KUKA KRL program: MyProgram_162().src

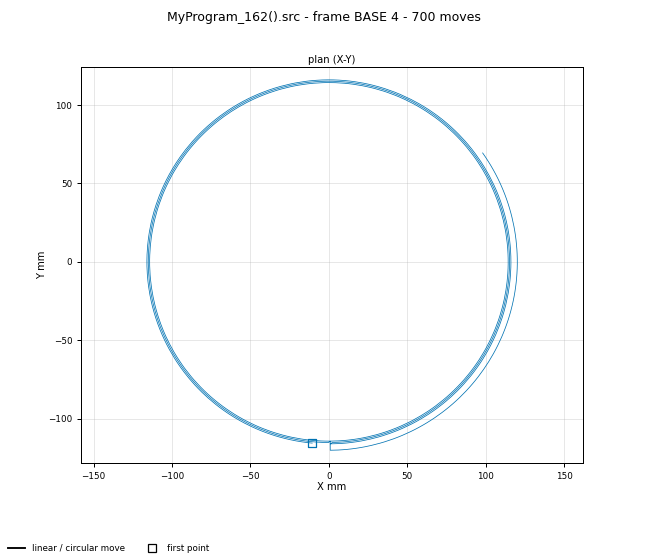
[picture p0: tool path of MyProgram_162().src in frame BASE 4, 700 of 700 moves have a stored position in this frame; points joined in program order, loops and branches not executed]
&ACCESS RVP
&REL 1
&PARAM TEMPLATE = C:\KRC\Roboter\Template\vorgabe
&PARAM EDITMASK = *
DEF MyProgram_162()
; ---- Setting reference (Base) ----
$BASE = BASE_DATA[4]

; --------------------------
; ---- Setting tool (TCP) ----
$TOOL = TOOL_DATA[3]
; --------------------------

$VEL.CP = VEL_APROX_PRINT
Startdeposition()
$VEL.CP = VEL_PRINT
LIN {X -10.6653,Y -115.559,Z 123,A -99.1684,B 24.9575,C -1.5067,E1 24.9847,E2 185.24} C_DIS
LIN {X -13.6922,Y -115.2397,Z 123,A -100.788,B 24.9577,C -1.5018,E1 24.9802,E2 186.8723} C_DIS
LIN {X -17.6034,Y -114.7073,Z 123,A -102.6994,B 24.9577,C -1.5039,E1 24.9749,E2 188.7803} C_DIS
LIN {X -20.9745,Y -114.1398,Z 123,A -104.185,B 24.9571,C -1.5133,E1 24.9709,E2 190.2451} C_DIS
LIN {X -25.0062,Y -113.3242,Z 123,A -106.7407,B 24.9583,C -1.4914,E1 24.9637,E2 192.8559} C_DIS
LIN {X -28.1463,Y -112.5871,Z 123,A -108.1226,B 24.9578,C -1.5013,E1 24.96,E2 194.216} C_DIS
LIN {X -31.7748,Y -111.6155,Z 123,A -109.9543,B 24.9576,C -1.5036,E1 24.9551,E2 196.0454} C_DIS
LIN {X -34.7534,Y -110.7249,Z 123,A -111.6242,B 24.9579,C -1.4989,E1 24.9506,E2 197.7293} C_DIS
LIN {X -38.9895,Y -109.306,Z 123,A -113.7372,B 24.9576,C -1.5047,E1 24.9451,E2 199.8326} C_DIS
LIN {X -42.4675,Y -108.0007,Z 123,A -115.4677,B 24.9572,C -1.5109,E1 24.9406,E2 201.5519} C_DIS
LIN {X -45.3067,Y -106.841,Z 123,A -117.0721,B 24.9574,C -1.5086,E1 24.9364,E2 203.1654} C_DIS
LIN {X -48.6937,Y -105.3407,Z 123,A -118.8003,B 24.957,C -1.515,E1 24.9321,E2 204.8826} C_DIS
LIN {X -53.8437,Y -102.8035,Z 123,A -121.6909,B 24.957,C -1.5162,E1 24.9249,E2 207.7782} C_DIS
LIN {X -57.1329,Y -101.0142,Z 123,A -124.0798,B 24.9581,C -1.4959,E1 24.9189,E2 210.2222} C_DIS
LIN {X -60.7707,Y -98.8681,Z 123,A -125.684,B 24.9568,C -1.5193,E1 24.9152,E2 211.7758} C_DIS
LIN {X -63.696,Y -97.0077,Z 123,A -127.252,B 24.9563,C -1.5281,E1 24.9115,E2 213.328} C_DIS
LIN {X -66.3521,Y -95.2106,Z 123,A -128.9266,B 24.9563,C -1.5268,E1 24.9077,E2 215.0111} C_DIS
LIN {X -69.3236,Y -93.0704,Z 123,A -130.8195,B 24.9563,C -1.5264,E1 24.9034,E2 216.9117} C_DIS
LIN {X -71.8676,Y -91.1191,Z 123,A -133.4324,B 24.9586,C -1.4866,E1 24.8975,E2 219.629} C_DIS
LIN {X -77.0205,Y -86.8086,Z 123,A -135.5024,B 24.9553,C -1.5447,E1 24.8934,E2 221.5689} C_DIS
LIN {X -81.0208,Y -83.0887,Z 123,A -138.4564,B 24.9556,C -1.5395,E1 24.8873,E2 224.5473} C_DIS
LIN {X -83.5609,Y -80.5308,Z 123,A -140.1615,B 24.9552,C -1.5465,E1 24.884,E2 226.2431} C_DIS
LIN {X -85.4663,Y -78.5057,Z 123,A -142.2929,B 24.9568,C -1.5184,E1 24.8799,E2 228.4508} C_DIS
LIN {X -88.8943,Y -74.604,Z 123,A -143.9688,B 24.9544,C -1.5609,E1 24.877,E2 230.0333} C_DIS
LIN {X -92.3379,Y -70.2979,Z 123,A -146.9806,B 24.9547,C -1.5555,E1 24.8717,E2 233.0722} C_DIS
LIN {X -94.5964,Y -67.2251,Z 123,A -148.7888,B 24.9542,C -1.5633,E1 24.8688,E2 234.8705} C_DIS
LIN {X -96.8103,Y -63.9955,Z 123,A -150.6696,B 24.9538,C -1.5704,E1 24.8658,E2 236.7437} C_DIS
LIN {X -98.2369,Y -61.784,Z 123,A -152.1414,B 24.954,C -1.5668,E1 24.8636,E2 238.2317} C_DIS
LIN {X -100.5513,Y -57.9404,Z 123,A -153.9732,B 24.9527,C -1.5884,E1 24.8611,E2 240.0214} C_DIS
LIN {X -101.7139,Y -55.8775,Z 123,A -155.4383,B 24.9533,C -1.5795,E1 24.859,E2 241.5155} C_DIS
LIN {X -103.2771,Y -52.9291,Z 123,A -157.0466,B 24.9529,C -1.5857,E1 24.857,E2 243.1175} C_DIS
LIN {X -104.6961,Y -50.0641,Z 123,A -158.8223,B 24.9531,C -1.5822,E1 24.8548,E2 244.9113} C_DIS
LIN {X -106.1854,Y -46.8231,Z 123,A -160.8908,B 24.9535,C -1.5748,E1 24.8524,E2 247.0087} C_DIS
LIN {X -107.7171,Y -43.1859,Z 123,A -162.4847,B 24.9523,C -1.5948,E1 24.8508,E2 248.5638} C_DIS
LIN {X -109.095,Y -39.5722,Z 123,A -164.3294,B 24.9518,C -1.6031,E1 24.849,E2 250.3991} C_DIS
LIN {X -110.3696,Y -35.8636,Z 123,A -166.2617,B 24.9515,C -1.6091,E1 24.8473,E2 252.328} C_DIS
LIN {X -111.5262,Y -32.0901,Z 123,A -168.0218,B 24.9507,C -1.6227,E1 24.8459,E2 254.0659} C_DIS
LIN {X -112.5763,Y -28.1905,Z 123,A -170.1776,B 24.9507,C -1.6223,E1 24.8444,E2 256.2354} C_DIS
LIN {X -113.2511,Y -25.3421,Z 123,A -171.5538,B 24.9502,C -1.6296,E1 24.8435,E2 257.6022} C_DIS
LIN {X -114.1339,Y -21.0071,Z 123,A -174.7127,B 24.9522,C -1.5975,E1 24.8418,E2 260.8563} C_DIS
LIN {X -115.0069,Y -15.5386,Z 123,A -176.6028,B 24.9496,C -1.6399,E1 24.8411,E2 262.6566} C_DIS
LIN {X -115.4108,Y -12.1655,Z 123,A -178.893,B 24.9508,C -1.6208,E1 24.8404,E2 265.006} C_DIS
LIN {X -115.7852,Y -7.8379,Z 123,A 178.8146,B 24.9508,C -1.6219,E1 24.84,E2 267.3096} C_DIS
LIN {X -116.0178,Y -2.8199,Z 123,A 176.9216,B 24.9488,C -1.6533,E1 24.8398,E2 269.1392} C_DIS
LIN {X -116.0475,Y 0.856,Z 123,A 174.7066,B 24.9494,C -1.6433,E1 24.8398,E2 271.3915} C_DIS
LIN {X -115.9508,Y 4.8049,Z 123,A 172.4484,B 24.9498,C -1.6374,E1 24.8401,E2 273.6772} C_DIS
LIN {X -115.6096,Y 10.1176,Z 123,A 170.5898,B 24.9473,C -1.6766,E1 24.8405,E2 275.4536} C_DIS
LIN {X -115.0956,Y 14.8542,Z 123,A 168.1879,B 24.947,C -1.6823,E1 24.8413,E2 277.8562} C_DIS
LIN {X -114.5033,Y 18.8864,Z 123,A 166.2109,B 24.9465,C -1.6902,E1 24.8421,E2 279.8261} C_DIS
LIN {X -113.9089,Y 22.1913,Z 123,A 164.4813,B 24.9463,C -1.6927,E1 24.843,E2 281.56} C_DIS
LIN {X -113.3762,Y 24.7683,Z 123,A 162.8897,B 24.9468,C -1.6852,E1 24.844,E2 283.1788} C_DIS
LIN {X -112.6272,Y 27.9821,Z 123,A 161.5978,B 24.9456,C -1.7039,E1 24.8448,E2 284.4338} C_DIS
LIN {X -111.4941,Y 32.2032,Z 123,A 159.3971,B 24.9453,C -1.7091,E1 24.8464,E2 286.6349} C_DIS
LIN {X -110.195,Y 36.4032,Z 123,A 156.9707,B 24.9455,C -1.7057,E1 24.8485,E2 289.0832} C_DIS
LIN {X -108.2506,Y 41.8313,Z 123,A 154.2761,B 24.9445,C -1.7207,E1 24.8511,E2 291.7574} C_DIS
LIN {X -106.9132,Y 45.1354,Z 123,A 152.6645,B 24.9438,C -1.7321,E1 24.8528,E2 293.3507} C_DIS
LIN {X -105.5414,Y 48.2602,Z 123,A 150.7928,B 24.9439,C -1.7297,E1 24.855,E2 295.2384} C_DIS
LIN {X -103.8814,Y 51.7333,Z 123,A 148.9469,B 24.9434,C -1.7376,E1 24.8572,E2 297.0754} C_DIS
LIN {X -101.8776,Y 55.5757,Z 123,A 146.1169,B 24.9448,C -1.7164,E1 24.8611,E2 299.971} C_DIS
LIN {X -99.431,Y 59.8444,Z 123,A 144.3767,B 24.9425,C -1.751,E1 24.8634,E2 301.6377} C_DIS
LIN {X -97.3709,Y 63.1413,Z 123,A 141.7758,B 24.944,C -1.7291,E1 24.8675,E2 304.3039} C_DIS
LIN {X -94.7272,Y 67.0417,Z 123,A 140.3014,B 24.9413,C -1.7698,E1 24.8697,E2 305.6885} C_DIS
LIN {X -91.4771,Y 71.4147,Z 123,A 137.3922,B 24.9414,C -1.7682,E1 24.8746,E2 308.6155} C_DIS
LIN {X -87.1641,Y 76.6172,Z 123,A 133.5732,B 24.9421,C -1.7574,E1 24.8816,E2 312.4776} C_DIS
LIN {X -84.599,Y 79.4396,Z 123,A 132.0333,B 24.9409,C -1.7761,E1 24.8844,E2 313.9799} C_DIS
LIN {X -82.0963,Y 82.026,Z 123,A 130.4546,B 24.94,C -1.7885,E1 24.8875,E2 315.5358} C_DIS
LIN {X -79.8971,Y 84.1676,Z 123,A 128.9268,B 24.9398,C -1.7916,E1 24.8905,E2 317.0624} C_DIS
LIN {X -77.5135,Y 86.3673,Z 123,A 127.1384,B 24.9401,C -1.7877,E1 24.8943,E2 318.8673} C_DIS
LIN {X -73.9241,Y 89.4593,Z 123,A 124.9854,B 24.9392,C -1.8006,E1 24.8988,E2 320.9979} C_DIS
LIN {X -72.0186,Y 90.9998,Z 123,A 123.6847,B 24.9393,C -1.7996,E1 24.9017,E2 322.306} C_DIS
LIN {X -69.5493,Y 92.9008,Z 123,A 122.1969,B 24.9389,C -1.8049,E1 24.9049,E2 323.7865} C_DIS
LIN {X -66.4177,Y 95.165,Z 123,A 120.2261,B 24.9389,C -1.8062,E1 24.9094,E2 325.761} C_DIS
LIN {X -64.3163,Y 96.5987,Z 123,A 118.456,B 24.9401,C -1.7876,E1 24.9137,E2 327.5813} C_DIS
LIN {X -61.0227,Y 98.7123,Z 123,A 116.9584,B 24.9387,C -1.8091,E1 24.9171,E2 329.0325} C_DIS
LIN {X -57.9117,Y 100.5678,Z 123,A 115.2449,B 24.9382,C -1.8154,E1 24.9212,E2 330.736} C_DIS
LIN {X -54.6063,Y 102.4019,Z 123,A 113.3425,B 24.9382,C -1.8171,E1 24.9259,E2 332.6397} C_DIS
LIN {X -51.6065,Y 103.9443,Z 123,A 111.7134,B 24.9378,C -1.8214,E1 24.9299,E2 334.263} C_DIS
LIN {X -49.021,Y 105.1883,Z 123,A 110.011,B 24.9385,C -1.8117,E1 24.9343,E2 335.9928} C_DIS
LIN {X -45.1475,Y 106.9081,Z 123,A 108.1625,B 24.9376,C -1.825,E1 24.939,E2 337.8141} C_DIS
LIN {X -42.56,Y 107.9644,Z 123,A 106.5783,B 24.938,C -1.8183,E1 24.9431,E2 339.4176} C_DIS
LIN {X -38.4699,Y 109.4884,Z 123,A 104.5881,B 24.9374,C -1.828,E1 24.9483,E2 341.3887} C_DIS
LIN {X -34.7829,Y 110.7157,Z 123,A 102.1474,B 24.9387,C -1.8084,E1 24.9549,E2 343.8804} C_DIS
LIN {X -30.8214,Y 111.8839,Z 123,A 100.7644,B 24.9367,C -1.8382,E1 24.9585,E2 345.1949} C_DIS
LIN {X -24.2525,Y 113.4886,Z 123,A 97.3058,B 24.9368,C -1.8362,E1 24.9679,E2 348.6629} C_DIS
LIN {X -21.2452,Y 114.0905,Z 123,A 94.6996,B 24.9399,C -1.7914,E1 24.9754,E2 351.3782} C_DIS
LIN {X -14.8714,Y 115.0933,Z 123,A 92.6352,B 24.9365,C -1.8408,E1 24.9807,E2 353.3269} C_DIS
LIN {X -11.5372,Y 115.4765,Z 123,A 90.862,B 24.9368,C -1.8367,E1 24.9857,E2 355.111} C_DIS
LIN {X -7.9886,Y 115.775,Z 123,A 89.1698,B 24.9365,C -1.8403,E1 24.9904,E2 356.7953} C_DIS
LIN {X -4.2713,Y 115.9737,Z 123,A 87.2428,B 24.9367,C -1.8371,E1 24.9958,E2 358.7304} C_DIS
LIN {X -0.6516,Y 116.0483,Z 123,A 85.579,B 24.9363,C -1.8429,E1 25.0004,E2 360.3805} C_DIS
LIN {X 2.8366,Y 116.0176,Z 123,A 83.7142,B 24.9368,C -1.8369,E1 25.0056,E2 362.2592} C_DIS
LIN {X 6.415,Y 115.8727,Z 123,A 82.0622,B 24.9364,C -1.8421,E1 25.0102,E2 363.8985} C_DIS
LIN {X 10.0554,Y 115.6153,Z 123,A 80.1581,B 24.9367,C -1.8375,E1 25.0155,E2 365.8124} C_DIS
LIN {X 13.4144,Y 115.2723,Z 123,A 78.5907,B 24.9364,C -1.8416,E1 25.0198,E2 367.3691} C_DIS
LIN {X 16.9015,Y 114.8143,Z 123,A 76.9179,B 24.9363,C -1.8439,E1 25.0244,E2 369.0349} C_DIS
LIN {X 22.1519,Y 113.9165,Z 123,A 73.8926,B 24.9375,C -1.8256,E1 25.0329,E2 372.1002} C_DIS
LIN {X 25.3525,Y 113.2488,Z 123,A 72.6719,B 24.9364,C -1.842,E1 25.0361,E2 373.2804} C_DIS
LIN {X 28.1703,Y 112.5796,Z 123,A 71.0663,B 24.937,C -1.8335,E1 25.0405,E2 374.904} C_DIS
LIN {X 31.8716,Y 111.5881,Z 123,A 69.1035,B 24.9373,C -1.829,E1 25.0458,E2 376.874} C_DIS
LIN {X 35.8448,Y 110.3757,Z 123,A 67.2411,B 24.9368,C -1.8358,E1 25.0507,E2 378.717} C_DIS
LIN {X 39.5647,Y 109.0977,Z 123,A 65.5874,B 24.9361,C -1.8468,E1 25.055,E2 380.3412} C_DIS
LIN {X 41.7509,Y 108.2819,Z 123,A 64.0219,B 24.9374,C -1.8273,E1 25.0592,E2 381.9496} C_DIS
LIN {X 45.319,Y 106.8358,Z 123,A 62.2201,B 24.9372,C -1.8297,E1 25.0638,E2 383.7415} C_DIS
LIN {X 52.4206,Y 103.537,Z 123,A 58.4693,B 24.9372,C -1.8301,E1 25.0733,E2 387.4816} C_DIS
LIN {X 57.4012,Y 100.8611,Z 123,A 55.567,B 24.9378,C -1.8212,E1 25.0804,E2 390.3965} C_DIS
LIN {X 60.4595,Y 99.0572,Z 123,A 53.8305,B 24.938,C -1.8194,E1 25.0845,E2 392.1321} C_DIS
LIN {X 63.7326,Y 96.9836,Z 123,A 51.8571,B 24.9384,C -1.8136,E1 25.0892,E2 394.1127} C_DIS
LIN {X 67.2845,Y 94.5539,Z 123,A 49.7895,B 24.9384,C -1.8125,E1 25.0939,E2 396.1757} C_DIS
LIN {X 69.3854,Y 93.024,Z 123,A 48.1836,B 24.9396,C -1.7956,E1 25.0976,E2 397.8157} C_DIS
LIN {X 72.0684,Y 90.9604,Z 123,A 46.557,B 24.9396,C -1.7945,E1 25.1011,E2 399.4389} C_DIS
LIN {X 74.6917,Y 88.8214,Z 123,A 45.1593,B 24.939,C -1.8037,E1 25.1041,E2 400.8096} C_DIS
LIN {X 77.4628,Y 86.4127,Z 123,A 43.4207,B 24.939,C -1.8035,E1 25.1077,E2 402.5419} C_DIS
LIN {X 80.3599,Y 83.7256,Z 123,A 41.486,B 24.9393,C -1.8001,E1 25.1116,E2 404.4764} C_DIS
LIN {X 82.6619,Y 81.4535,Z 123,A 39.6068,B 24.9404,C -1.7837,E1 25.1154,E2 406.3864} C_DIS
LIN {X 86.7428,Y 77.094,Z 123,A 36.8843,B 24.9401,C -1.7874,E1 25.1205,E2 409.0882} C_DIS
LIN {X 88.767,Y 74.7562,Z 123,A 35.3125,B 24.9405,C -1.7817,E1 25.1234,E2 410.6664} C_DIS
LIN {X 91.1283,Y 71.856,Z 123,A 33.585,B 24.9405,C -1.7828,E1 25.1263,E2 412.3833} C_DIS
LIN {X 93.4714,Y 68.7808,Z 123,A 31.6666,B 24.9408,C -1.7776,E1 25.1296,E2 414.3048} C_DIS
LIN {X 96.8913,Y 63.8727,Z 123,A 28.7323,B 24.9412,C -1.7709,E1 25.1342,E2 417.2404} C_DIS
LIN {X 99.1052,Y 60.3806,Z 123,A 26.9313,B 24.9408,C -1.7766,E1 25.1368,E2 419.0188} C_DIS
LIN {X 102.1738,Y 55.0296,Z 123,A 23.7699,B 24.9418,C -1.7628,E1 25.1412,E2 422.1963} C_DIS
LIN {X 105.2146,Y 48.9644,Z 123,A 20.4053,B 24.9424,C -1.7526,E1 25.1454,E2 425.567} C_DIS
LIN {X 106.7262,Y 45.5792,Z 123,A 18.5385,B 24.9429,C -1.7456,E1 25.1475,E2 427.4402} C_DIS
LIN {X 108.0181,Y 42.4232,Z 123,A 16.8907,B 24.9431,C -1.7423,E1 25.1492,E2 429.0866} C_DIS
LIN {X 109.3788,Y 38.7822,Z 123,A 14.9282,B 24.9436,C -1.7345,E1 25.1511,E2 431.0564} C_DIS
LIN {X 110.9984,Y 33.8711,Z 123,A 12.5513,B 24.9436,C -1.735,E1 25.1531,E2 433.4187} C_DIS
LIN {X 112.1204,Y 29.9461,Z 123,A 10.2332,B 24.9449,C -1.7146,E1 25.1549,E2 435.7716} C_DIS
LIN {X 113.1662,Y 25.7141,Z 123,A 8.2717,B 24.9448,C -1.7168,E1 25.1561,E2 437.7166} C_DIS
LIN {X 114.1323,Y 21.0161,Z 123,A 5.995,B 24.945,C -1.7136,E1 25.1573,E2 439.9875} C_DIS
LIN {X 114.678,Y 17.793,Z 123,A 4.3378,B 24.9454,C -1.7065,E1 25.1581,E2 441.6518} C_DIS
LIN {X 115.2213,Y 13.8498,Z 123,A 2.4673,B 24.9455,C -1.7046,E1 25.1588,E2 443.5156} C_DIS
LIN {X 115.5668,Y 10.5813,Z 123,A 0.8306,B 24.9459,C -1.6987,E1 25.1592,E2 445.1565} C_DIS
LIN {X 115.8416,Y 6.9777,Z 123,A -1.0576,B 24.9466,C -1.688,E1 25.1596,E2 447.0588} C_DIS
LIN {X 115.9975,Y 3.4945,Z 123,A -2.7088,B 24.9467,C -1.6858,E1 25.1597,E2 448.7055} C_DIS
LIN {X 116.0499,Y -0.4908,Z 123,A -4.6581,B 24.9471,C -1.6802,E1 25.1597,E2 450.6564} C_DIS
LIN {X 115.993,Y -3.6417,Z 123,A -6.2118,B 24.9474,C -1.6752,E1 25.1597,E2 452.2125} C_DIS
LIN {X 115.8011,Y -7.6013,Z 123,A -8.1306,B 24.9477,C -1.6706,E1 25.1594,E2 454.1307} C_DIS
LIN {X 115.5426,Y -10.843,Z 123,A -9.6833,B 24.9479,C -1.6679,E1 25.159,E2 455.6807} C_DIS
LIN {X 115.1957,Y -14.0682,Z 123,A -11.4618,B 24.9487,C -1.6543,E1 25.1584,E2 457.4807} C_DIS
LIN {X 114.3495,Y -19.8061,Z 123,A -14.2853,B 24.9492,C -1.6468,E1 25.1572,E2 460.3052} C_DIS
LIN {X 112.7554,Y -27.4564,Z 123,A -17.8097,B 24.949,C -1.6502,E1 25.1552,E2 463.8013} C_DIS
LIN {X 111.5256,Y -32.092,Z 123,A -20.3392,B 24.9499,C -1.6349,E1 25.1533,E2 466.3523} C_DIS
LIN {X 110.4511,Y -35.6117,Z 123,A -22.9008,B 24.9524,C -1.5941,E1 25.151,E2 468.9954} C_DIS
LIN {X 108.7581,Y -40.4935,Z 123,A -24.807,B 24.951,C -1.6163,E1 25.1493,E2 470.8387} C_DIS
LIN {X 107.4122,Y -43.9351,Z 123,A -26.5091,B 24.951,C -1.6164,E1 25.1475,E2 472.5311} C_DIS
LIN {X 106.4459,Y -46.2269,Z 123,A -28.2646,B 24.9528,C -1.5878,E1 25.1455,E2 474.3443} C_DIS
LIN {X 104.71,Y -50.0351,Z 123,A -29.7767,B 24.9516,C -1.6075,E1 25.1438,E2 475.8018} C_DIS
LIN {X 103.1305,Y -53.2159,Z 123,A -31.5677,B 24.952,C -1.6005,E1 25.1415,E2 477.5999} C_DIS
LIN {X 101.0864,Y -57.0036,Z 123,A -33.7107,B 24.9524,C -1.5933,E1 25.1386,E2 479.7486} C_DIS
LIN {X 98.3156,Y -61.658,Z 123,A -36.2905,B 24.9526,C -1.59,E1 25.1349,E2 482.3231} C_DIS
LIN {X 96.692,Y -64.1749,Z 123,A -37.9215,B 24.9533,C -1.5786,E1 25.1323,E2 483.9728} C_DIS
LIN {X 94.5646,Y -67.2696,Z 123,A -39.624,B 24.9532,C -1.5805,E1 25.1296,E2 485.6624} C_DIS
LIN {X 92.8107,Y -69.6692,Z 123,A -41.4058,B 24.9543,C -1.5618,E1 25.1266,E2 487.4799} C_DIS
LIN {X 90.753,Y -72.3308,Z 123,A -42.7436,B 24.9537,C -1.5724,E1 25.1243,E2 488.7865} C_DIS
LIN {X 86.1852,Y -77.717,Z 123,A -46.5937,B 24.9552,C -1.5463,E1 25.1172,E2 492.6807} C_DIS
LIN {X 83.7476,Y -80.3371,Z 123,A -47.9446,B 24.9543,C -1.5612,E1 25.1147,E2 493.9905} C_DIS
LIN {X 81.6168,Y -82.5005,Z 123,A -50.21,B 24.9566,C -1.5221,E1 25.11,E2 496.3388} C_DIS
LIN {X 77.7653,Y -86.1418,Z 123,A -52.5362,B 24.9562,C -1.5292,E1 25.1052,E2 498.6388} C_DIS
LIN {X 74.6982,Y -88.816,Z 123,A -54.107,B 24.9553,C -1.5449,E1 25.102,E2 500.1665} C_DIS
LIN {X 72.3115,Y -90.7683,Z 123,A -55.8805,B 24.9561,C -1.5299,E1 25.0981,E2 501.9688} C_DIS
LIN {X 68.7013,Y -93.5296,Z 123,A -57.7636,B 24.9555,C -1.5418,E1 25.0939,E2 503.8171} C_DIS
LIN {X 66.5136,Y -95.0983,Z 123,A -59.5656,B 24.9569,C -1.5172,E1 25.0897,E2 505.6708} C_DIS
LIN {X 63.2692,Y -97.2888,Z 123,A -61.1524,B 24.9562,C -1.5292,E1 25.0861,E2 507.224} C_DIS
LIN {X 58.7946,Y -100.0546,Z 123,A -64.0349,B 24.9572,C -1.5113,E1 25.0791,E2 510.1399} C_DIS
LIN {X 55.6291,Y -101.8487,Z 123,A -65.3622,B 24.9562,C -1.5296,E1 25.076,E2 511.4201} C_DIS
LIN {X 52.8234,Y -103.3311,Z 123,A -66.8836,B 24.9562,C -1.529,E1 25.0722,E2 512.9387} C_DIS
LIN {X 46.848,Y -106.1752,Z 123,A -70.2052,B 24.9566,C -1.5213,E1 25.0638,E2 516.27} C_DIS
LIN {X 43.6706,Y -107.5199,Z 123,A -71.9026,B 24.9568,C -1.5191,E1 25.0594,E2 517.9687} C_DIS
LIN {X 39.4119,Y -109.1534,Z 123,A -74.9392,B 24.9589,C -1.4806,E1 25.0512,E2 521.09} C_DIS
LIN {X 34.4921,Y -110.8059,Z 123,A -76.6276,B 24.9569,C -1.5168,E1 25.047,E2 522.6895} C_DIS
LIN {X 31.5546,Y -111.6779,Z 123,A -79.0047,B 24.9592,C -1.4763,E1 25.0403,E2 525.1586} C_DIS
LIN {X 26.4818,Y -112.9889,Z 123,A -80.5878,B 24.9568,C -1.5187,E1 25.0363,E2 526.6389} C_DIS
LIN {X 20.9624,Y -114.142,Z 123,A -83.6261,B 24.9576,C -1.5048,E1 25.0279,E2 529.7066} C_DIS
LIN {X 17.6866,Y -114.6945,Z 123,A -85.2438,B 24.9576,C -1.5046,E1 25.0235,E2 531.3231} C_DIS
LIN {X 13.9079,Y -115.2145,Z 123,A -87.056,B 24.9575,C -1.5065,E1 25.0185,E2 533.1293} C_DIS
LIN {X 10.5813,Y -115.5668,Z 123,A -88.7723,B 24.9577,C -1.5027,E1 25.0137,E2 534.8535} C_DIS
LIN {X 6.5999,Y -115.8625,Z 123,A -90.6749,B 24.9576,C -1.5049,E1 25.0084,E2 536.7502} C_DIS
LIN {X 3.4987,Y -115.9974,Z 123,A -92.2533,B 24.9577,C -1.5023,E1 25.004,E2 538.3342} C_DIS
LIN {X 0.8259,Y -116.0445,Z 123,A -93.2298,B 24.9569,C -1.5172,E1 25.0013,E2 539.2751} C_DIS
Enddeposition()
LIN {X 0.8259,Y -116.0445,Z 123,A -93.2298,B 24.9569,C -1.5172,E1 25.0013,E2 539.2751} C_DIS
Startdeposition()
$VEL.CP = VEL_PRINT
LIN {X 2.3314,Y -115.1543,Z 123,A -92.0357,B 24.9548,C -1.5524,E1 25.0049,E2 537.9978} C_DIS
LIN {X 5.8321,Y -115.0312,Z 123,A -90.2801,B 24.9548,C -1.5537,E1 25.0098,E2 536.2398} C_DIS
LIN {X 9.2842,Y -114.803,Z 123,A -88.6539,B 24.955,C -1.5503,E1 25.0143,E2 534.6225} C_DIS
LIN {X 12.0787,Y -114.5426,Z 123,A -87.2954,B 24.955,C -1.5493,E1 25.0181,E2 533.267} C_DIS
LIN {X 15.5256,Y -114.1286,Z 123,A -85.5808,B 24.955,C -1.5499,E1 25.0228,E2 531.5526} C_DIS
LIN {X 18.7354,Y -113.644,Z 123,A -83.8879,B 24.9547,C -1.5546,E1 25.0275,E2 529.8501} C_DIS
LIN {X 26.6527,Y -112.0535,Z 123,A -78.853,B 24.9517,C -1.6048,E1 25.0416,E2 524.703} C_DIS
LIN {X 32.6711,Y -110.4469,Z 123,A -77.1344,B 24.9553,C -1.545,E1 25.0458,E2 523.1288} C_DIS
LIN {X 36.1646,Y -109.3548,Z 123,A -74.9767,B 24.9543,C -1.5625,E1 25.0516,E2 520.9337} C_DIS
LIN {X 41.4613,Y -107.4586,Z 123,A -72.2545,B 24.9543,C -1.5627,E1 25.0588,E2 518.2166} C_DIS
LIN {X 45.8782,Y -105.6462,Z 123,A -69.8825,B 24.954,C -1.5661,E1 25.0649,E2 515.8422} C_DIS
LIN {X 49.7687,Y -103.8701,Z 123,A -68.0228,B 24.9546,C -1.5571,E1 25.0695,E2 514.0083} C_DIS
LIN {X 52.2474,Y -102.6458,Z 123,A -66.3315,B 24.9536,C -1.5739,E1 25.0738,E2 512.2819} C_DIS
LIN {X 55.1644,Y -101.1082,Z 123,A -64.7776,B 24.9536,C -1.5728,E1 25.0776,E2 510.735} C_DIS
LIN {X 57.9974,Y -99.5123,Z 123,A -62.5944,B 24.9519,C -1.602,E1 25.0831,E2 508.4894} C_DIS
LIN {X 61.2153,Y -97.5636,Z 123,A -61.2467,B 24.9532,C -1.5813,E1 25.0861,E2 507.1951} C_DIS
LIN {X 64.75,Y -95.2543,Z 123,A -59.1714,B 24.953,C -1.5843,E1 25.091,E2 505.1196} C_DIS
LIN {X 67.7817,Y -93.1217,Z 123,A -57.2697,B 24.9526,C -1.5908,E1 25.0953,E2 503.2091} C_DIS
LIN {X 70.324,Y -91.2165,Z 123,A -55.697,B 24.9524,C -1.5939,E1 25.0988,E2 501.6348} C_DIS
LIN {X 72.7159,Y -89.3217,Z 123,A -54.143,B 24.9521,C -1.5989,E1 25.1022,E2 500.0747} C_DIS
LIN {X 76.2027,Y -86.3677,Z 123,A -52.0079,B 24.9521,C -1.5977,E1 25.1067,E2 497.951} C_DIS
LIN {X 78.7583,Y -84.0421,Z 123,A -49.908,B 24.9508,C -1.6197,E1 25.1111,E2 495.8076} C_DIS
LIN {X 82.0112,Y -80.8708,Z 123,A -48.0104,B 24.9515,C -1.6082,E1 25.1148,E2 493.9453} C_DIS
LIN {X 84.7331,Y -78.0144,Z 123,A -46.011,B 24.9511,C -1.6149,E1 25.1186,E2 491.9387} C_DIS
LIN {X 87.0536,Y -75.4174,Z 123,A -44.0403,B 24.9502,C -1.6306,E1 25.1223,E2 489.9398} C_DIS
LIN {X 90.2153,Y -71.6041,Z 123,A -41.7943,B 24.9504,C -1.6269,E1 25.1262,E2 487.7129} C_DIS
LIN {X 92.6813,Y -68.3832,Z 123,A -39.8099,B 24.9502,C -1.6309,E1 25.1295,E2 485.7287} C_DIS
LIN {X 94.8891,Y -65.2861,Z 123,A -38.0501,B 24.9502,C -1.6299,E1 25.1323,E2 483.9798} C_DIS
LIN {X 96.3292,Y -63.1402,Z 123,A -36.7614,B 24.95,C -1.6338,E1 25.1343,E2 482.6885} C_DIS
LIN {X 98.7146,Y -59.3434,Z 123,A -34.5715,B 24.9497,C -1.6383,E1 25.1375,E2 480.499} C_DIS
LIN {X 99.9396,Y -57.2538,Z 123,A -33.3025,B 24.9493,C -1.6448,E1 25.1393,E2 479.221} C_DIS
LIN {X 101.3571,Y -54.7056,Z 123,A -31.8591,B 24.9491,C -1.6488,E1 25.1412,E2 477.7758} C_DIS
LIN {X 103.1084,Y -51.3283,Z 123,A -29.9074,B 24.9485,C -1.6573,E1 25.1437,E2 475.8144} C_DIS
LIN {X 104.8757,Y -47.614,Z 123,A -27.8111,B 24.948,C -1.6659,E1 25.1462,E2 473.7092} C_DIS
LIN {X 106.6754,Y -43.4312,Z 123,A -25.6989,B 24.948,C -1.6657,E1 25.1485,E2 471.6092} C_DIS
LIN {X 107.6962,Y -40.8344,Z 123,A -24.3607,B 24.9479,C -1.6677,E1 25.1498,E2 470.2738} C_DIS
LIN {X 109.0637,Y -37.028,Z 123,A -22.5714,B 24.9481,C -1.6634,E1 25.1515,E2 468.5045} C_DIS
LIN {X 109.9005,Y -34.4662,Z 123,A -20.9555,B 24.9471,C -1.6807,E1 25.1529,E2 466.857} C_DIS
LIN {X 110.9607,Y -30.8854,Z 123,A -19.2054,B 24.9471,C -1.6815,E1 25.1542,E2 465.115} C_DIS
LIN {X 111.84,Y -27.5278,Z 123,A -17.6828,B 24.9473,C -1.6774,E1 25.1553,E2 463.6108} C_DIS
LIN {X 113.0054,Y -22.2648,Z 123,A -14.8579,B 24.9463,C -1.6929,E1 25.157,E2 460.7659} C_DIS
LIN {X 113.4418,Y -19.9268,Z 123,A -12.8447,B 24.9435,C -1.7364,E1 25.158,E2 458.6619} C_DIS
LIN {X 114.1879,Y -15.0697,Z 123,A -10.7543,B 24.9441,C -1.7274,E1 25.1587,E2 456.6052} C_DIS
LIN {X 114.5879,Y -11.6464,Z 123,A -9.5474,B 24.9453,C -1.7087,E1 25.1591,E2 455.4493} C_DIS
LIN {X 114.8404,Y -8.8164,Z 123,A -7.9361,B 24.9444,C -1.7228,E1 25.1594,E2 453.8145} C_DIS
LIN {X 115.0733,Y -4.9043,Z 123,A -6.069,B 24.9442,C -1.7252,E1 25.1597,E2 451.9527} C_DIS
LIN {X 115.1712,Y -1.4134,Z 123,A -4.4562,B 24.9442,C -1.725,E1 25.1597,E2 450.3501} C_DIS
LIN {X 115.1652,Y 1.7413,Z 123,A -2.7721,B 24.9435,C -1.7356,E1 25.1597,E2 448.6511} C_DIS
LIN {X 115.0606,Y 5.1992,Z 123,A -1.0319,B 24.9431,C -1.7421,E1 25.1596,E2 446.9059} C_DIS
LIN {X 114.7967,Y 9.3624,Z 123,A 0.9125,B 24.9431,C -1.7426,E1 25.1592,E2 444.9718} C_DIS
LIN {X 114.5426,Y 12.0787,Z 123,A 2.2395,B 24.9429,C -1.7455,E1 25.1588,E2 443.6457} C_DIS
LIN {X 114.175,Y 15.1692,Z 123,A 3.9374,B 24.9421,C -1.7576,E1 25.1582,E2 441.9293} C_DIS
LIN {X 113.5049,Y 19.5675,Z 123,A 5.9766,B 24.9421,C -1.7564,E1 25.1573,E2 439.9051} C_DIS
LIN {X 111.9947,Y 26.8938,Z 123,A 10.6633,B 24.9383,C -1.8141,E1 25.1544,E2 435.1095} C_DIS
LIN {X 110.4889,Y 32.5293,Z 123,A 12.3442,B 24.9416,C -1.7649,E1 25.1532,E2 433.554} C_DIS
LIN {X 109.3174,Y 36.2757,Z 123,A 14.4251,B 24.9408,C -1.7769,E1 25.1514,E2 431.4568} C_DIS
LIN {X 108.6143,Y 38.3261,Z 123,A 15.5868,B 24.9403,C -1.7841,E1 25.1504,E2 430.2847} C_DIS
LIN {X 107.3068,Y 41.8478,Z 123,A 17.4964,B 24.9398,C -1.7916,E1 25.1485,E2 428.3681} C_DIS
LIN {X 106.0821,Y 44.8611,Z 123,A 19.0898,B 24.9396,C -1.7952,E1 25.1467,E2 426.7749} C_DIS
LIN {X 104.7653,Y 47.859,Z 123,A 20.6381,B 24.9396,C -1.7961,E1 25.145,E2 425.2329} C_DIS
LIN {X 103.097,Y 51.3513,Z 123,A 22.5826,B 24.9391,C -1.8025,E1 25.1426,E2 423.2838} C_DIS
LIN {X 101.7295,Y 54.0108,Z 123,A 24.0592,B 24.9389,C -1.8061,E1 25.1407,E2 421.8064} C_DIS
LIN {X 100.1351,Y 56.9137,Z 123,A 25.9287,B 24.9378,C -1.821,E1 25.1381,E2 419.9115} C_DIS
LIN {X 97.646,Y 61.0834,Z 123,A 28.1578,B 24.938,C -1.8187,E1 25.1349,E2 417.699} C_DIS
LIN {X 95.9683,Y 63.6875,Z 123,A 29.848,B 24.9372,C -1.8297,E1 25.1323,E2 415.9914} C_DIS
LIN {X 93.6657,Y 67.0274,Z 123,A 31.7492,B 24.9372,C -1.8294,E1 25.1292,E2 414.1002} C_DIS
LIN {X 91.1655,Y 70.3901,Z 123,A 33.7003,B 24.9373,C -1.8284,E1 25.126,E2 412.1609} C_DIS
LIN {X 89.0041,Y 73.1068,Z 123,A 35.6872,B 24.9362,C -1.8446,E1 25.1224,E2 410.145} C_DIS
LIN {X 85.9774,Y 76.641,Z 123,A 38.6674,B 24.9337,C -1.881,E1 25.1168,E2 407.092} C_DIS
LIN {X 82.109,Y 80.7718,Z 123,A 40.3086,B 24.937,C -1.8327,E1 25.1138,E2 405.572} C_DIS
LIN {X 79.2735,Y 83.5576,Z 123,A 42.5951,B 24.9358,C -1.8511,E1 25.1092,E2 403.2517} C_DIS
LIN {X 76.6345,Y 85.9833,Z 123,A 44.3915,B 24.9355,C -1.8553,E1 25.1054,E2 401.4524} C_DIS
LIN {X 73.4638,Y 88.7074,Z 123,A 47.2075,B 24.9328,C -1.8934,E1 25.0992,E2 398.5573} C_DIS
LIN {X 69.2974,Y 91.9989,Z 123,A 48.7143,B 24.9361,C -1.846,E1 25.0962,E2 397.1679} C_DIS
LIN {X 66.9579,Y 93.7153,Z 123,A 50.5132,B 24.9348,C -1.8647,E1 25.092,E2 395.3311} C_DIS
LIN {X 63.5999,Y 96.0261,Z 123,A 52.5279,B 24.9346,C -1.8675,E1 25.0873,E2 393.3167} C_DIS
LIN {X 60.2866,Y 98.1414,Z 123,A 54.5178,B 24.9343,C -1.8721,E1 25.0826,E2 391.3222} C_DIS
LIN {X 57.05,Y 100.0567,Z 123,A 56.4994,B 24.9338,C -1.8799,E1 25.0778,E2 389.3283} C_DIS
LIN {X 53.6291,Y 101.9305,Z 123,A 58.1553,B 24.9345,C -1.8697,E1 25.0738,E2 387.7013} C_DIS
LIN {X 50.8271,Y 103.3569,Z 123,A 59.8935,B 24.9338,C -1.8795,E1 25.0694,E2 385.9445} C_DIS
LIN {X 45.9483,Y 105.6157,Z 123,A 62.4797,B 24.9338,C -1.8786,E1 25.0628,E2 383.3668} C_DIS
LIN {X 42.1489,Y 107.1885,Z 123,A 64.4629,B 24.9338,C -1.878,E1 25.0577,E2 381.3896} C_DIS
LIN {X 39.4047,Y 108.2275,Z 123,A 65.976,B 24.9336,C -1.8817,E1 25.0537,E2 379.8709} C_DIS
LIN {X 36.4687,Y 109.2523,Z 123,A 67.4076,B 24.9339,C -1.8779,E1 25.05,E2 378.4511} C_DIS
LIN {X 33.395,Y 110.2321,Z 123,A 69.1185,B 24.9335,C -1.8839,E1 25.0454,E2 376.7293} C_DIS
LIN {X 30.1745,Y 111.155,Z 123,A 70.8376,B 24.9332,C -1.8874,E1 25.0408,E2 375.0047} C_DIS
LIN {X 25.2746,Y 112.3723,Z 123,A 73.9812,B 24.9311,C -1.9169,E1 25.032,E2 371.7955} C_DIS
LIN {X 20.6386,Y 113.3138,Z 123,A 76.1184,B 24.9317,C -1.9082,E1 25.0262,E2 369.6813} C_DIS
LIN {X 16.7655,Y 113.9524,Z 123,A 77.5933,B 24.9332,C -1.8876,E1 25.0223,E2 368.2565} C_DIS
LIN {X 13.4376,Y 114.3912,Z 123,A 79.2338,B 24.9332,C -1.8867,E1 25.0178,E2 366.6195} C_DIS
LIN {X 9.7512,Y 114.7656,Z 123,A 81.1862,B 24.9329,C -1.8917,E1 25.0123,E2 364.6564} C_DIS
LIN {X 6.014,Y 115.0211,Z 123,A 83.0353,B 24.9329,C -1.891,E1 25.0071,E2 362.8095} C_DIS
LIN {X 2.2685,Y 115.1555,Z 123,A 84.8238,B 24.9332,C -1.8875,E1 25.0022,E2 361.0297} C_DIS
LIN {X -1.388,Y 115.1714,Z 123,A 86.5786,B 24.9334,C -1.8843,E1 24.9973,E2 359.2825} C_DIS
LIN {X -4.7824,Y 115.0785,Z 123,A 88.3296,B 24.9333,C -1.8865,E1 24.9924,E2 357.526} C_DIS
LIN {X -8.4783,Y 114.8674,Z 123,A 90.2302,B 24.9332,C -1.8883,E1 24.9871,E2 355.6206} C_DIS
LIN {X -11.9162,Y 114.5597,Z 123,A 91.9091,B 24.9333,C -1.8858,E1 24.9824,E2 353.9466} C_DIS
LIN {X -15.1253,Y 114.1807,Z 123,A 94.1976,B 24.9313,C -1.9142,E1 24.9759,E2 351.589} C_DIS
LIN {X -19.8689,Y 113.4522,Z 123,A 95.7514,B 24.934,C -1.8766,E1 24.9719,E2 350.1232} C_DIS
LIN {X -23.768,Y 112.7003,Z 123,A 97.8985,B 24.9336,C -1.8822,E1 24.966,E2 347.9601} C_DIS
LIN {X -29.5268,Y 111.3299,Z 123,A 100.6829,B 24.9343,C -1.8726,E1 24.9585,E2 345.1949} C_DIS
LIN {X -34.1322,Y 110.0041,Z 123,A 102.9483,B 24.9348,C -1.8649,E1 24.9524,E2 342.9439} C_DIS
LIN {X -36.7898,Y 109.144,Z 123,A 104.6689,B 24.9339,C -1.8772,E1 24.9478,E2 341.1908} C_DIS
LIN {X -40.0594,Y 107.9886,Z 123,A 106.3653,B 24.9342,C -1.8738,E1 24.9433,E2 339.4993} C_DIS
LIN {X -43.1441,Y 106.7922,Z 123,A 107.9735,B 24.9345,C -1.8699,E1 24.9392,E2 337.8967} C_DIS
LIN {X -46.1205,Y 105.5406,Z 123,A 109.6043,B 24.9345,C -1.8686,E1 24.935,E2 336.2652} C_DIS
LIN {X -49.2401,Y 104.124,Z 123,A 111.4365,B 24.9344,C -1.8713,E1 24.9303,E2 334.4221} C_DIS
LIN {X -52.5191,Y 102.5069,Z 123,A 113.1695,B 24.9348,C -1.8648,E1 24.926,E2 332.7} C_DIS
LIN {X -56.1294,Y 100.5753,Z 123,A 115.1145,B 24.9353,C -1.8574,E1 24.9213,E2 330.7669} C_DIS
LIN {X -59.0882,Y 98.8676,Z 123,A 116.8219,B 24.9355,C -1.8546,E1 24.9172,E2 329.061} C_DIS
LIN {X -61.2144,Y 97.5641,Z 123,A 118.1593,B 24.9355,C -1.8563,E1 24.914,E2 327.7153} C_DIS
LIN {X -63.9403,Y 95.8017,Z 123,A 119.8177,B 24.9355,C -1.855,E1 24.9101,E2 326.0548} C_DIS
LIN {X -66.8643,Y 93.7821,Z 123,A 121.5472,B 24.9359,C -1.8498,E1 24.9062,E2 324.3316} C_DIS
LIN {X -69.9266,Y 91.5227,Z 123,A 123.2635,B 24.9366,C -1.8385,E1 24.9024,E2 322.6361} C_DIS
LIN {X -72.0436,Y 89.8665,Z 123,A 124.666,B 24.9366,C -1.8383,E1 24.8993,E2 321.229} C_DIS
LIN {X -76.2731,Y 86.3054,Z 123,A 127.7537,B 24.9361,C -1.8459,E1 24.8927,E2 318.111} C_DIS
LIN {X -79.4684,Y 83.3727,Z 123,A 129.8298,B 24.9367,C -1.8375,E1 24.8885,E2 316.0465} C_DIS
LIN {X -82.0118,Y 80.8702,Z 123,A 131.474,B 24.9374,C -1.8278,E1 24.8853,E2 314.4184} C_DIS
LIN {X -86.5419,Y 76.0033,Z 123,A 134.9836,B 24.9374,C -1.8276,E1 24.8786,E2 310.8937} C_DIS
LIN {X -89.914,Y 71.9851,Z 123,A 137.3788,B 24.9385,C -1.8119,E1 24.8744,E2 308.5248} C_DIS
LIN {X -93.4553,Y 67.3222,Z 123,A 140.5785,B 24.9382,C -1.8157,E1 24.8691,E2 305.3007} C_DIS
LIN {X -96.2955,Y 63.1914,Z 123,A 142.6334,B 24.9399,C -1.7908,E1 24.8659,E2 303.2949} C_DIS
LIN {X -97.6687,Y 61.047,Z 123,A 144.1881,B 24.9393,C -1.7989,E1 24.8635,E2 301.7131} C_DIS
LIN {X -99.7718,Y 57.5459,Z 123,A 146.4534,B 24.9391,C -1.8025,E1 24.8603,E2 299.4274} C_DIS
LIN {X -101.918,Y 53.6528,Z 123,A 148.4208,B 24.9402,C -1.786,E1 24.8577,E2 297.4888} C_DIS
LIN {X -103.2339,Y 51.0753,Z 123,A 149.8145,B 24.9406,C -1.7798,E1 24.856,E2 296.1025} C_DIS
LIN {X -104.7281,Y 47.9416,Z 123,A 151.5431,B 24.941,C -1.7746,E1 24.854,E2 294.3769} C_DIS
LIN {X -106.2495,Y 44.4639,Z 123,A 153.6237,B 24.9408,C -1.7767,E1 24.8517,E2 292.2799} C_DIS
LIN {X -109.1929,Y 36.6448,Z 123,A 157.5486,B 24.9423,C -1.7542,E1 24.8479,E2 288.3863} C_DIS
LIN {X -110.1441,Y 33.6806,Z 123,A 159.1722,B 24.9424,C -1.7523,E1 24.8465,E2 286.7579} C_DIS
LIN {X -110.8128,Y 31.4073,Z 123,A 160.5359,B 24.9422,C -1.7561,E1 24.8455,E2 285.3775} C_DIS
LIN {X -111.7546,Y 27.8776,Z 123,A 162.3489,B 24.9426,C -1.75,E1 24.8442,E2 283.5681} C_DIS
LIN {X -112.543,Y 24.4946,Z 123,A 164.0783,B 24.943,C -1.7446,E1 24.8432,E2 281.8417} C_DIS
LIN {X -113.1854,Y 21.3346,Z 123,A 165.5333,B 24.9437,C -1.7333,E1 24.8424,E2 280.4048} C_DIS
LIN {X -113.7394,Y 18.1542,Z 123,A 167.1329,B 24.944,C -1.7279,E1 24.8417,E2 278.8088} C_DIS
LIN {X -114.1152,Y 15.6194,Z 123,A 168.6483,B 24.9437,C -1.7334,E1 24.8411,E2 277.2711} C_DIS
LIN {X -114.6427,Y 11.1005,Z 123,A 170.7751,B 24.9445,C -1.7205,E1 24.8404,E2 275.1623} C_DIS
LIN {X -114.9071,Y 7.8916,Z 123,A 172.5882,B 24.9443,C -1.7239,E1 24.8401,E2 273.3303} C_DIS
LIN {X -115.0889,Y 4.5398,Z 123,A 174.8531,B 24.9431,C -1.7427,E1 24.8398,E2 271.007} C_DIS
LIN {X -115.1777,Y -0.4444,Z 123,A 176.4635,B 24.9459,C -1.6992,E1 24.8398,E2 269.4906} C_DIS
LIN {X -115.0022,Y -6.3554,Z 123,A 179.5965,B 24.946,C -1.6974,E1 24.8401,E2 266.3431} C_DIS
LIN {X -114.4259,Y -13.1406,Z 123,A -177.2873,B 24.9474,C -1.6754,E1 24.8409,E2 263.2604} C_DIS
LIN {X -114.1182,Y -15.5984,Z 123,A -175.775,B 24.9469,C -1.6828,E1 24.8414,E2 261.7217} C_DIS
LIN {X -113.6363,Y -18.7816,Z 123,A -173.8528,B 24.9464,C -1.6907,E1 24.8423,E2 259.769} C_DIS
LIN {X -112.7671,Y -23.4427,Z 123,A -171.8295,B 24.9478,C -1.6696,E1 24.8434,E2 257.7841} C_DIS
LIN {X -112.1366,Y -26.295,Z 123,A -170.3797,B 24.9481,C -1.665,E1 24.8443,E2 256.3369} C_DIS
LIN {X -111.3854,Y -29.3199,Z 123,A -168.732,B 24.9481,C -1.6641,E1 24.8454,E2 254.6816} C_DIS
LIN {X -110.6606,Y -31.9445,Z 123,A -167.2934,B 24.9481,C -1.6634,E1 24.8465,E2 253.2364} C_DIS
LIN {X -109.4457,Y -35.8851,Z 123,A -165.4023,B 24.9489,C -1.6506,E1 24.8481,E2 251.3649} C_DIS
LIN {X -108.3068,Y -39.187,Z 123,A -163.5861,B 24.9491,C -1.6486,E1 24.8498,E2 249.5431} C_DIS
LIN {X -107.1471,Y -42.2542,Z 123,A -161.8559,B 24.9491,C -1.6478,E1 24.8516,E2 247.8051} C_DIS
LIN {X -104.8479,Y -47.6757,Z 123,A -159.0789,B 24.95,C -1.6331,E1 24.8546,E2 245.0479} C_DIS
LIN {X -103.4596,Y -50.6199,Z 123,A -157.4591,B 24.9503,C -1.6285,E1 24.8566,E2 243.4303} C_DIS
LIN {X -102.4091,Y -52.7105,Z 123,A -156.1113,B 24.95,C -1.6328,E1 24.8583,E2 242.065} C_DIS
LIN {X -100.6677,Y -55.9639,Z 123,A -154.3456,B 24.9505,C -1.6249,E1 24.8607,E2 240.3089} C_DIS
LIN {X -99.1635,Y -58.5876,Z 123,A -152.8116,B 24.9507,C -1.622,E1 24.8628,E2 238.7737} C_DIS
LIN {X -97.5252,Y -61.2767,Z 123,A -151.2179,B 24.9509,C -1.619,E1 24.8652,E2 237.1791} C_DIS
LIN {X -95.2718,Y -64.7242,Z 123,A -149.1704,B 24.9512,C -1.6136,E1 24.8684,E2 235.1342} C_DIS
LIN {X -93.2854,Y -67.5582,Z 123,A -147.3757,B 24.9512,C -1.6123,E1 24.8713,E2 233.3338} C_DIS
LIN {X -91.2354,Y -70.2994,Z 123,A -145.5733,B 24.9512,C -1.6123,E1 24.8743,E2 231.5228} C_DIS
LIN {X -88.5785,Y -73.619,Z 123,A -143.6608,B 24.9521,C -1.5988,E1 24.8777,E2 229.6336} C_DIS
LIN {X -86.4223,Y -76.1402,Z 123,A -141.7273,B 24.9516,C -1.6068,E1 24.8813,E2 227.6723} C_DIS
LIN {X -83.3294,Y -79.5138,Z 123,A -139.6114,B 24.9523,C -1.595,E1 24.8853,E2 225.5753} C_DIS
LIN {X -80.8825,Y -81.9996,Z 123,A -137.992,B 24.9528,C -1.5864,E1 24.8885,E2 223.9693} C_DIS
LIN {X -77.7284,Y -84.9956,Z 123,A -135.8094,B 24.9531,C -1.5827,E1 24.8929,E2 221.7867} C_DIS
LIN {X -74.9282,Y -87.4744,Z 123,A -133.3244,B 24.9517,C -1.6055,E1 24.8983,E2 219.2377} C_DIS
LIN {X -71.645,Y -90.1831,Z 123,A -131.7984,B 24.9534,C -1.5765,E1 24.9015,E2 217.7751} C_DIS
LIN {X -68.9727,Y -92.2429,Z 123,A -130.0588,B 24.9534,C -1.5761,E1 24.9054,E2 216.0302} C_DIS
LIN {X -66.4739,Y -94.0606,Z 123,A -128.4595,B 24.9534,C -1.5761,E1 24.909,E2 214.4254} C_DIS
LIN {X -63.4026,Y -96.1562,Z 123,A -126.7141,B 24.9539,C -1.5686,E1 24.913,E2 212.6918} C_DIS
LIN {X -60.5421,Y -97.9841,Z 123,A -124.8126,B 24.9535,C -1.5751,E1 24.9176,E2 210.769} C_DIS
LIN {X -57.2915,Y -99.9179,Z 123,A -123.0883,B 24.9541,C -1.5657,E1 24.9217,E2 209.0619} C_DIS
LIN {X -53.9102,Y -101.7825,Z 123,A -121.2012,B 24.9543,C -1.5616,E1 24.9263,E2 207.1791} C_DIS
LIN {X -50.9994,Y -103.2715,Z 123,A -119.3721,B 24.9539,C -1.5683,E1 24.9309,E2 205.3293} C_DIS
LIN {X -47.2042,Y -105.0604,Z 123,A -117.4751,B 24.9545,C -1.5577,E1 24.9357,E2 203.4528} C_DIS
LIN {X -43.6586,Y -106.5828,Z 123,A -115.4457,B 24.9544,C -1.5604,E1 24.941,E2 201.4123} C_DIS
LIN {X -40.5141,Y -107.8174,Z 123,A -113.916,B 24.9549,C -1.5523,E1 24.9449,E2 199.8986} C_DIS
LIN {X -38.1422,Y -108.6788,Z 123,A -112.6182,B 24.9549,C -1.5531,E1 24.9483,E2 198.5964} C_DIS
LIN {X -34.6366,Y -109.8477,Z 123,A -110.6677,B 24.9546,C -1.5565,E1 24.9535,E2 196.6343} C_DIS
LIN {X -31.1796,Y -110.8774,Z 123,A -108.8545,B 24.9546,C -1.5561,E1 24.9584,E2 194.819} C_DIS
LIN {X -27.5998,Y -111.8224,Z 123,A -105.8432,B 24.9516,C -1.6068,E1 24.967,E2 191.6832} C_DIS
LIN {X -20.4348,Y -113.3505,Z 123,A -103.5548,B 24.9553,C -1.5452,E1 24.9728,E2 189.5387} C_DIS
LIN {X -17.5477,Y -113.8332,Z 123,A -102.0383,B 24.9551,C -1.5474,E1 24.977,E2 188.0155} C_DIS
LIN {X -13.9927,Y -114.3262,Z 123,A -100.2822,B 24.9552,C -1.5457,E1 24.9819,E2 186.262} C_DIS
LIN {X -11.0013,Y -114.6519,Z 123,A -98.683,B 24.955,C -1.5501,E1 24.9863,E2 184.6515} C_DIS
LIN {X -7.7573,Y -114.9162,Z 123,A -97.1231,B 24.9551,C -1.5475,E1 24.9907,E2 183.0972} C_DIS
LIN {X -3.991,Y -115.1095,Z 123,A -95.1733,B 24.9549,C -1.5509,E1 24.9961,E2 181.1388} C_DIS
LIN {X -0.2572,Y -115.1783,Z 123,A -93.4354,B 24.9552,C -1.546,E1 25.0009,E2 179.4127} C_DIS
LIN {X -0.2572,Y -115.1783,Z 123,A -93.4354,B 24.9552,C -1.546,E1 25.0009,E2 179.4127} C_DIS
Enddeposition()
LIN {X 0.8191,Y -114.3011,Z 123,A -93.4178,B 24.9557,C -1.5385,E1 25.0009,E2 179.4127} C_DIS
Startdeposition()
$VEL.CP = VEL_PRINT
LIN {X -2.0398,Y -114.2871,Z 123,A -94.999,B 24.956,C -1.5317,E1 24.9965,E2 181.01} C_DIS
LIN {X -5.0584,Y -114.1934,Z 123,A -96.5879,B 24.9562,C -1.5283,E1 24.992,E2 182.6073} C_DIS
LIN {X -8.7222,Y -113.9727,Z 123,A -98.2132,B 24.9557,C -1.5376,E1 24.9876,E2 184.2112} C_DIS
LIN {X -11.2056,Y -113.7569,Z 123,A -99.6025,B 24.9561,C -1.5316,E1 24.9837,E2 185.6155} C_DIS
LIN {X -14.2944,Y -113.4087,Z 123,A -101.252,B 24.9563,C -1.5279,E1 24.9791,E2 187.2748} C_DIS
LIN {X -17.5891,Y -112.944,Z 123,A -102.8742,B 24.9561,C -1.5303,E1 24.9746,E2 188.8927} C_DIS
LIN {X -21.3788,Y -112.2885,Z 123,A -104.7449,B 24.9559,C -1.5334,E1 24.9695,E2 190.7579} C_DIS
LIN {X -23.7508,Y -111.8123,Z 123,A -106.0731,B 24.9562,C -1.529,E1 24.9658,E2 192.0982} C_DIS
LIN {X -26.4385,Y -111.2077,Z 123,A -107.4849,B 24.9562,C -1.5283,E1 24.9619,E2 193.5134} C_DIS
LIN {X -29.4489,Y -110.4473,Z 123,A -108.9128,B 24.9559,C -1.5348,E1 24.9581,E2 194.9281} C_DIS
LIN {X -32.1403,Y -109.6943,Z 123,A -110.3156,B 24.9559,C -1.5356,E1 24.9544,E2 196.3312} C_DIS
LIN {X -34.5339,Y -108.966,Z 123,A -111.5722,B 24.9558,C -1.5364,E1 24.951,E2 197.5881} C_DIS
LIN {X -37.2949,Y -108.0515,Z 123,A -112.9834,B 24.9556,C -1.5396,E1 24.9473,E2 198.9943} C_DIS
LIN {X -40.1171,Y -107.0349,Z 123,A -114.5397,B 24.9556,C -1.5388,E1 24.9432,E2 200.5557} C_DIS
LIN {X -42.4408,Y -106.1366,Z 123,A -115.9442,B 24.9559,C -1.5334,E1 24.9395,E2 201.9761} C_DIS
LIN {X -45.0432,Y -105.0585,Z 123,A -117.3794,B 24.9559,C -1.5339,E1 24.9358,E2 203.4134} C_DIS
LIN {X -47.9137,Y -103.7791,Z 123,A -118.6467,B 24.9551,C -1.5487,E1 24.9327,E2 204.6487} C_DIS
LIN {X -50.4337,Y -102.5782,Z 123,A -120.1873,B 24.9553,C -1.5444,E1 24.9288,E2 206.2034} C_DIS
LIN {X -52.6528,Y -101.4587,Z 123,A -121.4361,B 24.9553,C -1.5459,E1 24.9256,E2 207.4522} C_DIS
LIN {X -55.117,Y -100.1414,Z 123,A -122.9567,B 24.9554,C -1.5427,E1 24.9219,E2 208.9845} C_DIS
LIN {X -57.8133,Y -98.6077,Z 123,A -124.3925,B 24.955,C -1.5499,E1 24.9184,E2 210.4074} C_DIS
LIN {X -60.2251,Y -97.1534,Z 123,A -125.9023,B 24.9551,C -1.548,E1 24.9148,E2 211.9265} C_DIS
LIN {X -62.8617,Y -95.4678,Z 123,A -127.296,B 24.9545,C -1.5577,E1 24.9116,E2 213.3016} C_DIS
LIN {X -64.9332,Y -94.0719,Z 123,A -128.6486,B 24.9547,C -1.5556,E1 24.9085,E2 214.6637} C_DIS
LIN {X -67.2167,Y -92.4541,Z 123,A -130.0567,B 24.9545,C -1.5578,E1 24.9053,E2 216.0715} C_DIS
LIN {X -69.6479,Y -90.6361,Z 123,A -131.6236,B 24.9545,C -1.5587,E1 24.9018,E2 217.6421} C_DIS
LIN {X -72.1145,Y -88.6862,Z 123,A -133.2404,B 24.9545,C -1.5599,E1 24.8982,E2 219.2619} C_DIS
LIN {X -75.08,Y -86.19,Z 123,A -135.1558,B 24.9541,C -1.5648,E1 24.8942,E2 221.173} C_DIS
LIN {X -77.2756,Y -84.227,Z 123,A -136.6053,B 24.9539,C -1.5689,E1 24.8912,E2 222.6187} C_DIS
LIN {X -79.3286,Y -82.2963,Z 123,A -138.052,B 24.9538,C -1.5705,E1 24.8883,E2 224.0676} C_DIS
LIN {X -81.8134,Y -79.8296,Z 123,A -139.9507,B 24.9539,C -1.5683,E1 24.8845,E2 225.9794} C_DIS
LIN {X -84.2382,Y -77.2633,Z 123,A -141.592,B 24.9534,C -1.5775,E1 24.8814,E2 227.6061} C_DIS
LIN {X -85.9871,Y -75.3123,Z 123,A -142.9243,B 24.9532,C -1.5798,E1 24.8789,E2 228.939} C_DIS
LIN {X -88.0115,Y -72.9363,Z 123,A -144.5241,B 24.9532,C -1.582,E1 24.8761,E2 230.5408} C_DIS
LIN {X -90.452,Y -69.8867,Z 123,A -146.1761,B 24.9521,C -1.5992,E1 24.8733,E2 232.1598} C_DIS
LIN {X -91.8161,Y -68.088,Z 123,A -147.5592,B 24.9525,C -1.5917,E1 24.8709,E2 233.5673} C_DIS
LIN {X -93.4887,Y -65.7722,Z 123,A -148.9741,B 24.9523,C -1.596,E1 24.8686,E2 234.9788} C_DIS
LIN {X -95.2091,Y -63.2542,Z 123,A -150.3996,B 24.9518,C -1.6041,E1 24.8664,E2 236.3921} C_DIS
LIN {X -96.566,Y -61.1651,Z 123,A -151.9046,B 24.9522,C -1.5971,E1 24.8641,E2 237.9216} C_DIS
LIN {X -98.7669,Y -57.5436,Z 123,A -154.0429,B 24.9519,C -1.6022,E1 24.861,E2 240.0587} C_DIS
LIN {X -100.293,Y -54.8376,Z 123,A -155.4951,B 24.9514,C -1.6107,E1 24.8591,E2 241.4982} C_DIS
LIN {X -101.5411,Y -52.4918,Z 123,A -156.7585,B 24.951,C -1.6171,E1 24.8574,E2 242.753} C_DIS
LIN {X -102.857,Y -49.8627,Z 123,A -158.1797,B 24.9506,C -1.6234,E1 24.8557,E2 244.1669} C_DIS
LIN {X -103.9261,Y -47.5977,Z 123,A -159.8274,B 24.9514,C -1.6113,E1 24.8537,E2 245.8525} C_DIS
LIN {X -105.6571,Y -43.6188,Z 123,A -161.9128,B 24.9508,C -1.6212,E1 24.8514,E2 247.9258} C_DIS
LIN {X -107.2535,Y -39.529,Z 123,A -163.9848,B 24.95,C -1.6329,E1 24.8494,E2 249.9817} C_DIS
LIN {X -108.1894,Y -36.8903,Z 123,A -165.3973,B 24.9498,C -1.6367,E1 24.8481,E2 251.393} C_DIS
LIN {X -108.9691,Y -34.5242,Z 123,A -166.817,B 24.95,C -1.6337,E1 24.8469,E2 252.8281} C_DIS
LIN {X -110.171,Y -30.4715,Z 123,A -168.9014,B 24.9495,C -1.6415,E1 24.8453,E2 254.9058} C_DIS
LIN {X -110.9567,Y -27.4673,Z 123,A -170.2126,B 24.9486,C -1.6561,E1 24.8444,E2 256.1899} C_DIS
LIN {X -111.5956,Y -24.744,Z 123,A -171.626,B 24.9484,C -1.66,E1 24.8435,E2 257.6022} C_DIS
LIN {X -112.1194,Y -22.2567,Z 123,A -173.0456,B 24.9484,C -1.6583,E1 24.8427,E2 259.0345} C_DIS
LIN {X -112.6798,Y -19.2119,Z 123,A -174.4705,B 24.9478,C -1.6682,E1 24.842,E2 260.4441} C_DIS
LIN {X -113.1153,Y -16.455,Z 123,A -176.0198,B 24.9479,C -1.6667,E1 24.8413,E2 262.0062} C_DIS
LIN {X -113.4835,Y -13.6873,Z 123,A -177.4469,B 24.9477,C -1.6701,E1 24.8408,E2 263.4337} C_DIS
LIN {X -113.7883,Y -10.8656,Z 123,A -178.7187,B 24.9471,C -1.6806,E1 24.8405,E2 264.688} C_DIS
LIN {X -113.9982,Y -8.4026,Z 123,A 179.7143,B 24.9476,C -1.6717,E1 24.8401,E2 266.2858} C_DIS
LIN {X -114.1889,Y -5.1626,Z 123,A 178.4008,B 24.9465,C -1.6893,E1 24.8399,E2 267.5651} C_DIS
LIN {X -114.2794,Y -2.4604,Z 123,A 176.8508,B 24.9467,C -1.686,E1 24.8399,E2 269.1323} C_DIS
LIN {X -114.2994,Y 1.3242,Z 123,A 174.8392,B 24.9467,C -1.6877,E1 24.8399,E2 271.1522} C_DIS
LIN {X -114.2281,Y 4.2504,Z 123,A 173.5034,B 24.946,C -1.6976,E1 24.8399,E2 272.4722} C_DIS
LIN {X -114.0702,Y 7.3371,Z 123,A 171.9414,B 24.9457,C -1.7022,E1 24.8402,E2 274.0327} C_DIS
LIN {X -113.8831,Y 9.8379,Z 123,A 170.6863,B 24.9454,C -1.7063,E1 24.8405,E2 275.2855} C_DIS
LIN {X -113.6081,Y 12.6235,Z 123,A 169.1466,B 24.9454,C -1.7055,E1 24.8409,E2 276.8363} C_DIS
LIN {X -113.2653,Y 15.3991,Z 123,A 167.7341,B 24.9452,C -1.7097,E1 24.8414,E2 278.2475} C_DIS
LIN {X -112.8546,Y 18.1663,Z 123,A 166.3212,B 24.945,C -1.7138,E1 24.842,E2 279.6589} C_DIS
LIN {X -112.3179,Y 21.2259,Z 123,A 164.8686,B 24.9444,C -1.723,E1 24.8428,E2 281.0982} C_DIS
LIN {X -111.8304,Y 23.6672,Z 123,A 163.4982,B 24.9444,C -1.7222,E1 24.8435,E2 282.4787} C_DIS
LIN {X -111.1682,Y 26.6005,Z 123,A 162.1818,B 24.9436,C -1.7345,E1 24.8444,E2 283.7732} C_DIS
LIN {X -110.4459,Y 29.4539,Z 123,A 160.6137,B 24.9436,C -1.7356,E1 24.8455,E2 285.348} C_DIS
LIN {X -109.6958,Y 32.1354,Z 123,A 159.2027,B 24.9433,C -1.7394,E1 24.8465,E2 286.7579} C_DIS
LIN {X -108.9708,Y 34.5189,Z 123,A 157.9445,B 24.9431,C -1.743,E1 24.8476,E2 288.015} C_DIS
LIN {X -108.0428,Y 37.3199,Z 123,A 156.4738,B 24.9427,C -1.748,E1 24.8489,E2 289.482} C_DIS
LIN {X -107.0138,Y 40.1728,Z 123,A 154.9337,B 24.9425,C -1.752,E1 24.8504,E2 291.0214} C_DIS
LIN {X -106.1291,Y 42.4592,Z 123,A 153.6949,B 24.9422,C -1.7554,E1 24.8516,E2 292.259} C_DIS
LIN {X -105.0552,Y 45.0508,Z 123,A 152.1585,B 24.9423,C -1.7546,E1 24.8533,E2 293.806} C_DIS
LIN {X -103.7903,Y 47.8897,Z 123,A 150.8456,B 24.9413,C -1.769,E1 24.8548,E2 295.0915} C_DIS
LIN {X -102.5863,Y 50.4173,Z 123,A 149.2923,B 24.9415,C -1.7673,E1 24.8567,E2 296.6574} C_DIS
LIN {X -101.2154,Y 53.1147,Z 123,A 147.8273,B 24.941,C -1.7739,E1 24.8586,E2 298.1145} C_DIS
LIN {X -100.1285,Y 55.1402,Z 123,A 146.4933,B 24.9413,C -1.7701,E1 24.8604,E2 299.4647} C_DIS
LIN {X -98.5938,Y 57.8369,Z 123,A 145.182,B 24.9403,C -1.7843,E1 24.8622,E2 300.7489} C_DIS
LIN {X -97.1499,Y 60.2308,Z 123,A 143.6315,B 24.9405,C -1.7824,E1 24.8644,E2 302.3118} C_DIS
LIN {X -95.7947,Y 62.3659,Z 123,A 142.2144,B 24.9406,C -1.7801,E1 24.8666,E2 303.7416} C_DIS
LIN {X -94.0244,Y 65.0016,Z 123,A 140.7619,B 24.9399,C -1.7901,E1 24.8688,E2 305.1775} C_DIS
LIN {X -92.4283,Y 67.252,Z 123,A 139.368,B 24.9397,C -1.7934,E1 24.8711,E2 306.5702} C_DIS
LIN {X -90.6282,Y 69.6581,Z 123,A 137.8116,B 24.9396,C -1.7955,E1 24.8737,E2 308.129} C_DIS
LIN {X -88.7137,Y 72.0805,Z 123,A 136.2206,B 24.9394,C -1.7979,E1 24.8765,E2 309.7217} C_DIS
LIN {X -86.231,Y 75.033,Z 123,A 134.2966,B 24.939,C -1.8034,E1 24.88,E2 311.6416} C_DIS
LIN {X -83.7734,Y 77.7699,Z 123,A 132.3934,B 24.9389,C -1.8056,E1 24.8836,E2 313.5478} C_DIS
LIN {X -81.7177,Y 79.9265,Z 123,A 130.8763,B 24.9387,C -1.8084,E1 24.8865,E2 315.0649} C_DIS
LIN {X -79.4149,Y 82.2131,Z 123,A 129.2863,B 24.9383,C -1.8138,E1 24.8897,E2 316.6487} C_DIS
LIN {X -76.6807,Y 84.7709,Z 123,A 127.3166,B 24.9383,C -1.8145,E1 24.8938,E2 318.6247} C_DIS
LIN {X -73.996,Y 87.1225,Z 123,A 125.5776,B 24.9379,C -1.8206,E1 24.8974,E2 320.356} C_DIS
LIN {X -71.2649,Y 89.3715,Z 123,A 123.7731,B 24.9377,C -1.8232,E1 24.9013,E2 322.161} C_DIS
LIN {X -69.1867,Y 90.9909,Z 123,A 122.5657,B 24.9372,C -1.8306,E1 24.904,E2 323.3553} C_DIS
LIN {X -66.9455,Y 92.6524,Z 123,A 121.1605,B 24.937,C -1.8332,E1 24.9071,E2 324.7591} C_DIS
LIN {X -64.4164,Y 94.4266,Z 123,A 119.6008,B 24.9368,C -1.8359,E1 24.9107,E2 326.3178} C_DIS
LIN {X -62.3414,Y 95.8109,Z 123,A 118.3382,B 24.9367,C -1.8378,E1 24.9137,E2 327.5799} C_DIS
LIN {X -59.6882,Y 97.4842,Z 123,A 116.9088,B 24.9361,C -1.8466,E1 24.917,E2 328.9929} C_DIS
LIN {X -57.5508,Y 98.7627,Z 123,A 115.4004,B 24.9367,C -1.8383,E1 24.9207,E2 330.5257} C_DIS
LIN {X -54.8438,Y 100.2896,Z 123,A 113.9515,B 24.9362,C -1.8455,E1 24.9242,E2 331.9617} C_DIS
LIN {X -52.646,Y 101.4622,Z 123,A 112.6975,B 24.936,C -1.8473,E1 24.9273,E2 333.2147} C_DIS
LIN {X -49.8676,Y 102.8547,Z 123,A 111.2704,B 24.9355,C -1.8552,E1 24.9308,E2 334.6268} C_DIS
LIN {X -47.1847,Y 104.1123,Z 123,A 109.6932,B 24.9355,C -1.8538,E1 24.9348,E2 336.2114} C_DIS
LIN {X -44.4873,Y 105.2929,Z 123,A 108.1832,B 24.9355,C -1.8545,E1 24.9387,E2 337.7231} C_DIS
LIN {X -41.1229,Y 106.654,Z 123,A 106.2257,B 24.9358,C -1.8513,E1 24.9438,E2 339.6925} C_DIS
LIN {X -38.2094,Y 107.7306,Z 123,A 104.7786,B 24.9353,C -1.8579,E1 24.9476,E2 341.127} C_DIS
LIN {X -35.5611,Y 108.6336,Z 123,A 103.3284,B 24.9353,C -1.8576,E1 24.9514,E2 342.5805} C_DIS
LIN {X -33.1653,Y 109.3903,Z 123,A 102.1111,B 24.9351,C -1.8608,E1 24.9547,E2 343.7924} C_DIS
LIN {X -30.3536,Y 110.2029,Z 123,A 100.5614,B 24.9352,C -1.8589,E1 24.9589,E2 345.3489} C_DIS
LIN {X -27.442,Y 110.9629,Z 123,A 99.2679,B 24.9345,C -1.8694,E1 24.9623,E2 346.6194} C_DIS
LIN {X -24.7296,Y 111.5988,Z 123,A 97.8705,B 24.9345,C -1.8706,E1 24.9661,E2 348.0158} C_DIS
LIN {X -22.3027,Y 112.1106,Z 123,A 96.4818,B 24.9348,C -1.8656,E1 24.9699,E2 349.4181} C_DIS
LIN {X -19.26,Y 112.6718,Z 123,A 95.0587,B 24.9343,C -1.8721,E1 24.9738,E2 350.8271} C_DIS
LIN {X -16.275,Y 113.1409,Z 123,A 93.6373,B 24.9339,C -1.8771,E1 24.9777,E2 352.2379} C_DIS
LIN {X -13.6845,Y 113.4839,Z 123,A 92.1005,B 24.9346,C -1.8683,E1 24.982,E2 353.7967} C_DIS
LIN {X -9.7914,Y 113.8872,Z 123,A 90.1373,B 24.9346,C -1.8693,E1 24.9875,E2 355.7587} C_DIS
LIN {X -6.6915,Y 114.1099,Z 123,A 88.5775,B 24.9345,C -1.8698,E1 24.9918,E2 357.3177} C_DIS
LIN {X -4.2032,Y 114.2301,Z 123,A 87.2129,B 24.9348,C -1.8653,E1 24.9957,E2 358.6932} C_DIS
LIN {X -1.4024,Y 114.2988,Z 123,A 85.7822,B 24.9348,C -1.8645,E1 24.9997,E2 360.1259} C_DIS
LIN {X 1.9386,Y 114.289,Z 123,A 84.3194,B 24.9342,C -1.8739,E1 25.0037,E2 361.5665} C_DIS
LIN {X 4.2143,Y 114.2297,Z 123,A 83.1066,B 24.9344,C -1.8709,E1 25.0071,E2 362.7862} C_DIS
LIN {X 7.4941,Y 114.0596,Z 123,A 81.5187,B 24.9342,C -1.8734,E1 25.0115,E2 364.3673} C_DIS
LIN {X 9.8058,Y 113.8861,Z 123,A 80.2972,B 24.9344,C -1.8707,E1 25.0149,E2 365.5946} C_DIS
LIN {X 12.5934,Y 113.6116,Z 123,A 78.7462,B 24.9349,C -1.8642,E1 25.0193,E2 367.16} C_DIS
LIN {X 15.5598,Y 113.2425,Z 123,A 77.3101,B 24.9347,C -1.8666,E1 25.0232,E2 368.5893} C_DIS
LIN {X 18.7619,Y 112.755,Z 123,A 75.8463,B 24.9342,C -1.873,E1 25.0272,E2 370.0366} C_DIS
LIN {X 21.2713,Y 112.3092,Z 123,A 74.5027,B 24.9345,C -1.8696,E1 25.0309,E2 371.3866} C_DIS
LIN {X 23.6899,Y 111.8256,Z 123,A 73.1536,B 24.9349,C -1.8641,E1 25.0346,E2 372.747} C_DIS
LIN {X 26.4285,Y 111.2102,Z 123,A 71.8589,B 24.9346,C -1.8682,E1 25.0381,E2 374.0303} C_DIS
LIN {X 29.4374,Y 110.4504,Z 123,A 70.3046,B 24.9346,C -1.8673,E1 25.0423,E2 375.5843} C_DIS
LIN {X 32.1448,Y 109.693,Z 123,A 68.8977,B 24.9346,C -1.8664,E1 25.0461,E2 376.991} C_DIS
LIN {X 34.528,Y 108.9679,Z 123,A 67.6509,B 24.9348,C -1.8655,E1 25.0494,E2 378.2377} C_DIS
LIN {X 37.1866,Y 108.0895,Z 123,A 66.249,B 24.9348,C -1.8644,E1 25.0531,E2 379.6395} C_DIS
LIN {X 40.1094,Y 107.0378,Z 123,A 64.6892,B 24.935,C -1.8628,E1 25.0572,E2 381.1997} C_DIS
LIN {X 42.451,Y 106.1324,Z 123,A 63.3073,B 24.9354,C -1.8561,E1 25.0609,E2 382.5944} C_DIS
LIN {X 45.0783,Y 105.0432,Z 123,A 61.9086,B 24.9354,C -1.8557,E1 25.0644,E2 383.9907} C_DIS
LIN {X 48.8907,Y 103.3241,Z 123,A 59.8149,B 24.9356,C -1.8534,E1 25.0697,E2 386.0847} C_DIS
LIN {X 51.7861,Y 101.9018,Z 123,A 58.4223,B 24.9351,C -1.8612,E1 25.0732,E2 387.4549} C_DIS
LIN {X 53.8766,Y 100.8141,Z 123,A 57.0431,B 24.9358,C -1.8509,E1 25.0766,E2 388.8548} C_DIS
LIN {X 56.6106,Y 99.303,Z 123,A 55.5744,B 24.9356,C -1.8529,E1 25.0802,E2 390.3142} C_DIS
LIN {X 59.2413,Y 97.7557,Z 123,A 53.9951,B 24.936,C -1.8485,E1 25.084,E2 391.8992} C_DIS
LIN {X 62.351,Y 95.8046,Z 123,A 52.1033,B 24.9363,C -1.8432,E1 25.0885,E2 393.7972} C_DIS
LIN {X 64.9291,Y 94.0747,Z 123,A 50.6659,B 24.9361,C -1.8459,E1 25.0917,E2 395.2234} C_DIS
LIN {X 67.2115,Y 92.4579,Z 123,A 49.2691,B 24.9363,C -1.8437,E1 25.0949,E2 396.6206} C_DIS
LIN {X 69.384,Y 90.8394,Z 123,A 47.7574,B 24.9369,C -1.8344,E1 25.0983,E2 398.1488} C_DIS
LIN {X 72.1326,Y 88.6714,Z 123,A 46.0644,B 24.9369,C -1.8339,E1 25.102,E2 399.8366} C_DIS
LIN {X 75.0837,Y 86.1868,Z 123,A 44.2043,B 24.9369,C -1.8334,E1 25.1059,E2 401.6907} C_DIS
LIN {X 77.2859,Y 84.2175,Z 123,A 42.7673,B 24.9371,C -1.8324,E1 25.1089,E2 403.1243} C_DIS
LIN {X 79.3262,Y 82.2985,Z 123,A 41.338,B 24.9373,C -1.8283,E1 25.1118,E2 404.5574} C_DIS
LIN {X 81.5239,Y 80.1226,Z 123,A 39.6751,B 24.9379,C -1.8198,E1 25.1151,E2 406.2332} C_DIS
LIN {X 83.9124,Y 77.6184,Z 123,A 38.1143,B 24.9377,C -1.8238,E1 25.1181,E2 407.7779} C_DIS
LIN {X 85.9975,Y 75.3004,Z 123,A 36.5048,B 24.938,C -1.8181,E1 25.1211,E2 409.3936} C_DIS
LIN {X 88.0206,Y 72.9254,Z 123,A 34.9178,B 24.9384,C -1.8133,E1 25.1239,E2 410.9845} C_DIS
LIN {X 90.4502,Y 69.8891,Z 123,A 33.2969,B 24.9377,C -1.8235,E1 25.1267,E2 412.5737} C_DIS
LIN {X 91.8117,Y 68.0941,Z 123,A 31.9263,B 24.9386,C -1.8097,E1 25.129,E2 413.9705} C_DIS
LIN {X 93.4503,Y 65.8271,Z 123,A 30.5319,B 24.9388,C -1.8065,E1 25.1313,E2 415.3657} C_DIS
LIN {X 95.2153,Y 63.2447,Z 123,A 29.1131,B 24.9386,C -1.8093,E1 25.1335,E2 416.7709} C_DIS
LIN {X 96.7777,Y 60.8265,Z 123,A 27.5463,B 24.9393,C -1.7998,E1 25.1359,E2 418.3521} C_DIS
LIN {X 98.0603,Y 58.7394,Z 123,A 26.3203,B 24.9395,C -1.7966,E1 25.1376,E2 419.5795} C_DIS
LIN {X 99.6149,Y 56.0598,Z 123,A 24.7753,B 24.9398,C -1.7927,E1 25.1398,E2 421.1256} C_DIS
LIN {X 100.9543,Y 53.6105,Z 123,A 23.5215,B 24.9396,C -1.7955,E1 25.1414,E2 422.3662} C_DIS
LIN {X 102.0967,Y 51.4047,Z 123,A 22.0361,B 24.9406,C -1.781,E1 25.1433,E2 423.8781} C_DIS
LIN {X 103.3344,Y 48.869,Z 123,A 20.7396,B 24.9405,C -1.7823,E1 25.1449,E2 425.1643} C_DIS
LIN {X 104.6237,Y 46.0406,Z 123,A 19.0976,B 24.941,C -1.774,E1 25.1468,E2 426.8171} C_DIS
LIN {X 105.906,Y 43.0074,Z 123,A 17.5004,B 24.9412,C -1.7716,E1 25.1485,E2 428.4111} C_DIS
LIN {X 107.2525,Y 39.5317,Z 123,A 15.6941,B 24.9414,C -1.7689,E1 25.1503,E2 430.2137} C_DIS
LIN {X 108.1886,Y 36.8929,Z 123,A 14.2945,B 24.9416,C -1.7649,E1 25.1516,E2 431.615} C_DIS
LIN {X 108.972,Y 34.5148,Z 123,A 12.9057,B 24.9423,C -1.7549,E1 25.1528,E2 433.0195} C_DIS
LIN {X 109.8035,Y 31.7692,Z 123,A 11.6326,B 24.9421,C -1.7581,E1 25.1538,E2 434.2778} C_DIS
LIN {X 110.616,Y 28.8084,Z 123,A 10.1003,B 24.9424,C -1.7536,E1 25.1549,E2 435.8118} C_DIS
LIN {X 111.247,Y 26.2702,Z 123,A 8.7409,B 24.9428,C -1.7473,E1 25.1558,E2 437.1782} C_DIS
LIN {X 111.8207,Y 23.7124,Z 123,A 7.3005,B 24.9434,C -1.7373,E1 25.1566,E2 438.6339} C_DIS
LIN {X 112.3765,Y 20.9215,Z 123,A 5.9569,B 24.9434,C -1.7366,E1 25.1573,E2 439.9712} C_DIS
LIN {X 112.8552,Y 18.1629,Z 123,A 4.564,B 24.9437,C -1.7326,E1 25.158,E2 441.3654} C_DIS
LIN {X 113.3373,Y 14.8453,Z 123,A 3.0823,B 24.9435,C -1.7365,E1 25.1585,E2 442.8292} C_DIS
LIN {X 113.6435,Y 12.2882,Z 123,A 1.7261,B 24.944,C -1.7293,E1 25.159,E2 444.1943} C_DIS
LIN {X 113.9975,Y 8.4118,Z 123,A -0.325,B 24.9447,C -1.7183,E1 25.1594,E2 446.2591} C_DIS
LIN {X 114.1965,Y 4.9861,Z 123,A -1.9493,B 24.9447,C -1.7172,E1 25.1597,E2 447.8763} C_DIS
LIN {X 114.2882,Y 1.9812,Z 123,A -3.4885,B 24.9451,C -1.7108,E1 25.1597,E2 449.4215} C_DIS
LIN {X 114.2988,Y -1.4027,Z 123,A -5.2149,B 24.9456,C -1.7038,E1 25.1597,E2 451.154} C_DIS
LIN {X 114.2302,Y -4.2018,Z 123,A -6.4952,B 24.9456,C -1.705,E1 25.1597,E2 452.4241} C_DIS
LIN {X 114.0656,Y -7.4052,Z 123,A -8.1423,B 24.946,C -1.6979,E1 25.1594,E2 454.078} C_DIS
LIN {X 113.82,Y -10.522,Z 123,A -9.4942,B 24.9457,C -1.7029,E1 25.1591,E2 455.4103} C_DIS
LIN {X 113.5913,Y -12.7675,Z 123,A -10.8569,B 24.9466,C -1.6883,E1 25.1587,E2 456.7992} C_DIS
LIN {X 113.2557,Y -15.4672,Z 123,A -12.2241,B 24.9469,C -1.6837,E1 25.1582,E2 458.1692} C_DIS
LIN {X 112.8501,Y -18.1932,Z 123,A -13.6017,B 24.9471,C -1.6794,E1 25.1576,E2 459.5489} C_DIS
LIN {X 112.3196,Y -21.2173,Z 123,A -15.0397,B 24.9471,C -1.6791,E1 25.1568,E2 460.9791} C_DIS
LIN {X 111.8242,Y -23.696,Z 123,A -16.3932,B 24.9477,C -1.6709,E1 25.1561,E2 462.344} C_DIS
LIN {X 111.2134,Y -26.4152,Z 123,A -17.6794,B 24.9477,C -1.6716,E1 25.1553,E2 463.6212} C_DIS
LIN {X 110.4482,Y -29.4455,Z 123,A -19.2257,B 24.9479,C -1.6675,E1 25.1542,E2 465.1682} C_DIS
LIN {X 109.6301,Y -32.3567,Z 123,A -20.6551,B 24.9479,C -1.6667,E1 25.1531,E2 466.5913} C_DIS
LIN {X 108.9146,Y -34.6926,Z 123,A -21.868,B 24.9482,C -1.6633,E1 25.1521,E2 467.8053} C_DIS
LIN {X 108.095,Y -37.1705,Z 123,A -23.2525,B 24.9486,C -1.6556,E1 25.1508,E2 469.2001} C_DIS
LIN {X 107.0335,Y -40.1207,Z 123,A -24.8087,B 24.9489,C -1.6514,E1 25.1493,E2 470.7575} C_DIS
LIN {X 106.1346,Y -42.4457,Z 123,A -26.1775,B 24.9495,C -1.642,E1 25.1479,E2 472.141} C_DIS
LIN {X 105.0504,Y -45.0618,Z 123,A -27.571,B 24.9497,C -1.6388,E1 25.1464,E2 473.5345} C_DIS
LIN {X 103.7873,Y -47.896,Z 123,A -28.8665,B 24.9492,C -1.6461,E1 25.1449,E2 474.8056} C_DIS
LIN {X 102.5849,Y -50.4201,Z 123,A -30.397,B 24.9499,C -1.6359,E1 25.1431,E2 476.3521} C_DIS
LIN {X 101.3326,Y -52.8922,Z 123,A -31.6517,B 24.9497,C -1.6379,E1 25.1415,E2 477.5952} C_DIS
LIN {X 100.1464,Y -55.1078,Z 123,A -33.1399,B 24.9506,C -1.6235,E1 25.1395,E2 479.1095} C_DIS
LIN {X 98.6125,Y -57.8053,Z 123,A -34.4463,B 24.9502,C -1.6305,E1 25.1377,E2 480.3927} C_DIS
LIN {X 97.1685,Y -60.2011,Z 123,A -35.9665,B 24.9508,C -1.621,E1 25.1354,E2 481.9277} C_DIS
LIN {X 95.8042,Y -62.3516,Z 123,A -37.3493,B 24.9513,C -1.6124,E1 25.1333,E2 483.3238} C_DIS
LIN {X 94.0748,Y -64.929,Z 123,A -38.7832,B 24.9513,C -1.6137,E1 25.1311,E2 484.7476} C_DIS
LIN {X 92.4584,Y -67.2108,Z 123,A -40.1765,B 24.9514,C -1.6101,E1 25.1288,E2 486.1425} C_DIS
LIN {X 90.6412,Y -69.6412,Z 123,A -41.7315,B 24.9518,C -1.6044,E1 25.1262,E2 487.7036} C_DIS
LIN {X 88.6995,Y -72.098,Z 123,A -43.3275,B 24.9521,C -1.599,E1 25.1234,E2 489.3049} C_DIS
LIN {X 86.1891,Y -75.081,Z 123,A -45.2309,B 24.9523,C -1.5962,E1 25.12,E2 491.2062} C_DIS
LIN {X 84.2252,Y -77.2776,Z 123,A -46.6654,B 24.9523,C -1.5943,E1 25.1173,E2 492.6388} C_DIS
LIN {X 82.2986,Y -79.3261,Z 123,A -48.0964,B 24.9526,C -1.5898,E1 25.1145,E2 494.0742} C_DIS
LIN {X 79.8105,Y -81.8318,Z 123,A -49.884,B 24.953,C -1.5846,E1 25.111,E2 495.8666} C_DIS
LIN {X 77.6779,Y -83.8578,Z 123,A -51.2898,B 24.953,C -1.5842,E1 25.1081,E2 497.2675} C_DIS
LIN {X 75.3137,Y -85.9859,Z 123,A -52.921,B 24.9533,C -1.5788,E1 25.1047,E2 498.9049} C_DIS
LIN {X 72.9357,Y -88.012,Z 123,A -54.5146,B 24.9536,C -1.574,E1 25.1013,E2 500.5038} C_DIS
LIN {X 69.8851,Y -90.4533,Z 123,A -56.1416,B 24.9529,C -1.5849,E1 25.0978,E2 502.0991} C_DIS
LIN {X 68.0904,Y -91.8144,Z 123,A -57.5096,B 24.9537,C -1.5715,E1 25.0947,E2 503.4938} C_DIS
LIN {X 65.8247,Y -93.4521,Z 123,A -58.9061,B 24.9539,C -1.5688,E1 25.0915,E2 504.8918} C_DIS
LIN {X 63.2632,Y -95.2031,Z 123,A -60.548,B 24.9543,C -1.5617,E1 25.0877,E2 506.5449} C_DIS
LIN {X 60.6703,Y -96.8753,Z 123,A -61.9232,B 24.954,C -1.5665,E1 25.0845,E2 507.9043} C_DIS
LIN {X 58.7388,Y -98.0607,Z 123,A -63.1234,B 24.9543,C -1.5614,E1 25.0816,E2 509.1128} C_DIS
LIN {X 56.0568,Y -99.6166,Z 123,A -64.6724,B 24.9545,C -1.5588,E1 25.0778,E2 510.6632} C_DIS
LIN {X 53.6052,Y -100.9571,Z 123,A -65.9279,B 24.9542,C -1.5629,E1 25.0748,E2 511.9055} C_DIS
LIN {X 51.3971,Y -102.1006,Z 123,A -67.4232,B 24.955,C -1.5496,E1 25.071,E2 513.4282} C_DIS
LIN {X 48.4346,Y -103.5366,Z 123,A -68.744,B 24.9543,C -1.5618,E1 25.0677,E2 514.7167} C_DIS
LIN {X 46.0329,Y -104.6271,Z 123,A -70.273,B 24.955,C -1.5504,E1 25.0638,E2 516.2688} C_DIS
LIN {X 43.2637,Y -105.8016,Z 123,A -71.7713,B 24.955,C -1.5486,E1 25.0599,E2 517.7678} C_DIS
LIN {X 39.5017,Y -107.2634,Z 123,A -73.7913,B 24.9552,C -1.546,E1 25.0546,E2 519.7898} C_DIS
LIN {X 36.7937,Y -108.222,Z 123,A -75.1992,B 24.9552,C -1.5455,E1 25.0509,E2 521.1959} C_DIS
LIN {X 33.18,Y -109.3859,Z 123,A -77.1573,B 24.9555,C -1.5408,E1 25.0457,E2 523.1617} C_DIS
LIN {X 30.4406,Y -110.1794,Z 123,A -78.659,B 24.9558,C -1.536,E1 25.0416,E2 524.6722} C_DIS
LIN {X 27.4633,Y -110.9577,Z 123,A -79.9483,B 24.9552,C -1.5456,E1 25.0382,E2 525.9367} C_DIS
LIN {X 24.7629,Y -111.5915,Z 123,A -81.3504,B 24.9553,C -1.5438,E1 25.0344,E2 527.3412} C_DIS
LIN {X 21.4041,Y -112.2836,Z 123,A -83.2626,B 24.9559,C -1.5337,E1 25.0291,E2 529.2748} C_DIS
LIN {X 18.143,Y -112.8583,Z 123,A -84.9665,B 24.9561,C -1.5305,E1 25.0244,E2 530.9847} C_DIS
LIN {X 15.3738,Y -113.2688,Z 123,A -86.3683,B 24.9561,C -1.5296,E1 25.0205,E2 532.3875} C_DIS
LIN {X 12.2882,Y -113.6435,Z 123,A -87.8103,B 24.9559,C -1.5338,E1 25.0165,E2 533.8185} C_DIS
LIN {X 9.1737,Y -113.9366,Z 123,A -89.4057,B 24.956,C -1.5318,E1 25.0121,E2 535.4177} C_DIS
LIN {X 6.0373,Y -114.1461,Z 123,A -91.0011,B 24.9561,C -1.5302,E1 25.0076,E2 537.0162} C_DIS
LIN {X 2.4911,Y -114.2788,Z 123,A -92.5884,B 24.9557,C -1.538,E1 25.0033,E2 538.5847} C_DIS
LIN {X 0.8191,Y -114.3011,Z 123,A -93.417,B 24.9557,C -1.5382,E1 25.001,E2 539.4127} C_DIS
Enddeposition()
LIN {X 0.8495,Y -120.1163,Z 124,A -93.1002,B 24.9602,C -1.458,E1 25.0013,E2 539.2859} C_DIS
Startdeposition()
$VEL.CP = VEL_PRINT
LIN {X 2.9479,Y -120.0854,Z 124,A -91.735,B 24.9592,C -1.4753,E1 25.0052,E2 537.88} C_DIS
LIN {X 5.8941,Y -119.9769,Z 124,A -90.3296,B 24.9592,C -1.4758,E1 25.0092,E2 536.4739} C_DIS
LIN {X 8.8367,Y -119.7961,Z 124,A -88.9248,B 24.9592,C -1.4763,E1 25.0131,E2 535.0684} C_DIS
LIN {X 11.774,Y -119.5431,Z 124,A -87.5201,B 24.9592,C -1.477,E1 25.017,E2 533.6628} C_DIS
LIN {X 14.7042,Y -119.2182,Z 124,A -86.1158,B 24.9591,C -1.4778,E1 25.0209,E2 532.2578} C_DIS
LIN {X 17.6255,Y -118.8214,Z 124,A -84.7116,B 24.9591,C -1.4787,E1 25.0248,E2 530.8527} C_DIS
LIN {X 20.5362,Y -118.3531,Z 124,A -83.3075,B 24.959,C -1.4796,E1 25.0286,E2 529.4478} C_DIS
LIN {X 23.4346,Y -117.8134,Z 124,A -81.7389,B 24.9585,C -1.4886,E1 25.033,E2 527.8599} C_DIS
LIN {X 27.0074,Y -117.0438,Z 124,A -80.1641,B 24.9588,C -1.4822,E1 25.0372,E2 526.3023} C_DIS
LIN {X 29.9303,Y -116.3306,Z 124,A -78.745,B 24.9588,C -1.4829,E1 25.0411,E2 524.8836} C_DIS
LIN {X 32.7179,Y -115.5776,Z 124,A -77.3581,B 24.9587,C -1.4849,E1 25.0448,E2 523.4943} C_DIS
LIN {X 35.5445,Y -114.7398,Z 124,A -75.9423,B 24.9586,C -1.487,E1 25.0486,E2 522.0761} C_DIS
LIN {X 38.4071,Y -113.8136,Z 124,A -74.5368,B 24.9586,C -1.4874,E1 25.0523,E2 520.6723} C_DIS
LIN {X 41.1317,Y -112.8576,Z 124,A -73.1374,B 24.9584,C -1.4902,E1 25.056,E2 519.269} C_DIS
LIN {X 43.9454,Y -111.792,Z 124,A -71.7193,B 24.9584,C -1.4914,E1 25.0597,E2 517.8513} C_DIS
LIN {X 46.6786,Y -110.6786,Z 124,A -70.3166,B 24.9582,C -1.4932,E1 25.0633,E2 516.4475} C_DIS
LIN {X 49.3778,Y -109.501,Z 124,A -68.9291,B 24.9582,C -1.4946,E1 25.0669,E2 515.0602} C_DIS
LIN {X 51.9956,Y -108.2825,Z 124,A -67.5433,B 24.958,C -1.4972,E1 25.0704,E2 513.6718} C_DIS
LIN {X 54.6373,Y -106.9739,Z 124,A -66.142,B 24.9579,C -1.4993,E1 25.0739,E2 512.2693} C_DIS
LIN {X 57.2462,Y -105.6008,Z 124,A -64.7281,B 24.9577,C -1.5021,E1 25.0773,E2 510.8528} C_DIS
LIN {X 59.8205,Y -104.1641,Z 124,A -63.3403,B 24.9577,C -1.5038,E1 25.0807,E2 509.4651} C_DIS
LIN {X 62.4106,Y -102.6332,Z 124,A -61.9108,B 24.9575,C -1.5062,E1 25.0841,E2 508.0343} C_DIS
LIN {X 64.8595,Y -101.1033,Z 124,A -60.5394,B 24.9574,C -1.5086,E1 25.0874,E2 506.6617} C_DIS
LIN {X 67.3714,Y -99.4472,Z 124,A -59.11,B 24.9572,C -1.5112,E1 25.0907,E2 505.2309} C_DIS
LIN {X 69.7916,Y -97.7639,Z 124,A -57.7231,B 24.9572,C -1.5132,E1 25.0939,E2 503.8441} C_DIS
LIN {X 72.1214,Y -96.058,Z 124,A -56.3391,B 24.9569,C -1.5165,E1 25.097,E2 502.4574} C_DIS
LIN {X 74.5046,Y -94.2216,Z 124,A -54.9104,B 24.9568,C -1.5193,E1 25.1001,E2 501.0273} C_DIS
LIN {X 76.7479,Y -92.4035,Z 124,A -53.527,B 24.9566,C -1.5227,E1 25.1031,E2 499.6412} C_DIS
LIN {X 78.9925,Y -90.4922,Z 124,A -52.1404,B 24.9564,C -1.525,E1 25.1061,E2 498.2546} C_DIS
LIN {X 81.234,Y -88.4853,Z 124,A -50.6953,B 24.9562,C -1.5289,E1 25.109,E2 496.8061} C_DIS
LIN {X 83.3812,Y -86.4652,Z 124,A -49.3264,B 24.9562,C -1.5304,E1 25.1118,E2 495.4392} C_DIS
LIN {X 85.478,Y -84.3928,Z 124,A -47.9276,B 24.9559,C -1.5336,E1 25.1146,E2 494.039} C_DIS
LIN {X 87.4819,Y -82.3138,Z 124,A -46.5445,B 24.9557,C -1.5373,E1 25.1172,E2 492.6529} C_DIS
LIN {X 89.516,Y -80.097,Z 124,A -45.1174,B 24.9555,C -1.5406,E1 25.1199,E2 491.2244} C_DIS
LIN {X 91.4154,Y -77.9221,Z 124,A -43.7346,B 24.9553,C -1.5445,E1 25.1224,E2 489.8387} C_DIS
LIN {X 93.3029,Y -75.6519,Z 124,A -42.3485,B 24.9552,C -1.5472,E1 25.1249,E2 488.4527} C_DIS
LIN {X 95.1658,Y -73.2948,Z 124,A -40.9225,B 24.9549,C -1.5507,E1 25.1274,E2 487.0251} C_DIS
LIN {X 96.9358,Y -70.9372,Z 124,A -39.5375,B 24.9548,C -1.5536,E1 25.1297,E2 485.64} C_DIS
LIN {X 98.613,Y -68.5866,Z 124,A -38.1556,B 24.9545,C -1.5577,E1 25.1319,E2 484.2553} C_DIS
LIN {X 100.2998,Y -66.0953,Z 124,A -36.7288,B 24.9543,C -1.5613,E1 25.1341,E2 482.8268} C_DIS
LIN {X 101.8596,Y -63.6653,Z 124,A -35.3601,B 24.9541,C -1.5649,E1 25.1361,E2 481.4567} C_DIS
LIN {X 103.4221,Y -61.0942,Z 124,A -33.9338,B 24.9539,C -1.5686,E1 25.1382,E2 480.0288} C_DIS
LIN {X 104.8608,Y -58.5906,Z 124,A -32.5521,B 24.9536,C -1.5729,E1 25.1401,E2 478.6442} C_DIS
LIN {X 106.2953,Y -55.946,Z 124,A -31.1391,B 24.9535,C -1.5761,E1 25.142,E2 477.2311} C_DIS
LIN {X 107.6363,Y -53.3205,Z 124,A -29.7418,B 24.9532,C -1.5799,E1 25.1437,E2 475.8323} C_DIS
LIN {X 108.9124,Y -50.6629,Z 124,A -28.3574,B 24.953,C -1.5831,E1 25.1454,E2 474.4478} C_DIS
LIN {X 110.0987,Y -48.0303,Z 124,A -26.9763,B 24.9528,C -1.5876,E1 25.1469,E2 473.0637} C_DIS
LIN {X 111.2443,Y -45.3139,Z 124,A -25.5794,B 24.9525,C -1.5915,E1 25.1484,E2 471.6654} C_DIS
LIN {X 112.3228,Y -42.5702,Z 124,A -24.1694,B 24.9523,C -1.5961,E1 25.1498,E2 470.2524} C_DIS
LIN {X 113.3538,Y -39.7437,Z 124,A -22.7698,B 24.9521,C -1.5988,E1 25.1512,E2 468.8541} C_DIS
LIN {X 114.2764,Y -37.0075,Z 124,A -21.3757,B 24.9518,C -1.604,E1 25.1524,E2 467.4556} C_DIS
LIN {X 115.1674,Y -34.1338,Z 124,A -19.9631,B 24.9516,C -1.6075,E1 25.1535,E2 466.0429} C_DIS
LIN {X 115.9704,Y -31.2972,Z 124,A -18.5339,B 24.9512,C -1.6131,E1 25.1546,E2 464.6085} C_DIS
LIN {X 116.8711,Y -27.7551,Z 124,A -16.7935,B 24.9509,C -1.6186,E1 25.1557,E2 462.8654} C_DIS
LIN {X 117.517,Y -24.8785,Z 124,A -15.4386,B 24.9508,C -1.6206,E1 25.1565,E2 461.5136} C_DIS
LIN {X 118.0921,Y -21.987,Z 124,A -14.0421,B 24.9505,C -1.6247,E1 25.1573,E2 460.1157} C_DIS
LIN {X 118.5962,Y -19.0823,Z 124,A -12.6454,B 24.9503,C -1.6288,E1 25.1579,E2 458.7175} C_DIS
LIN {X 119.0288,Y -16.166,Z 124,A -11.2466,B 24.95,C -1.633,E1 25.1585,E2 457.3169} C_DIS
LIN {X 119.3896,Y -13.2401,Z 124,A -9.7984,B 24.9496,C -1.6397,E1 25.1589,E2 455.8615} C_DIS
LIN {X 119.6786,Y -10.3061,Z 124,A -8.456,B 24.9496,C -1.6411,E1 25.1593,E2 454.5237} C_DIS
LIN {X 119.8955,Y -7.3659,Z 124,A -7.0596,B 24.9493,C -1.6453,E1 25.1595,E2 453.1259} C_DIS
LIN {X 120.0402,Y -4.4213,Z 124,A -5.6629,B 24.949,C -1.6494,E1 25.1597,E2 451.7277} C_DIS
LIN {X 120.1125,Y -1.4741,Z 124,A -4.1265,B 24.9483,C -1.6605,E1 25.1597,E2 450.1744} C_DIS
LIN {X 120.0995,Y 2.1807,Z 124,A -2.5354,B 24.9484,C -1.6586,E1 25.1597,E2 448.5971} C_DIS
LIN {X 120.0098,Y 5.1274,Z 124,A -1.139,B 24.9482,C -1.6627,E1 25.1596,E2 447.1993} C_DIS
LIN {X 119.8437,Y 8.1315,Z 124,A 0.2736,B 24.948,C -1.6663,E1 25.1594,E2 445.7868} C_DIS
LIN {X 119.6081,Y 11.0702,Z 124,A 1.67,B 24.9477,C -1.6703,E1 25.159,E2 444.3891} C_DIS
LIN {X 119.3074,Y 13.942,Z 124,A 3.0638,B 24.9474,C -1.6756,E1 25.1586,E2 442.9911} C_DIS
LIN {X 118.9193,Y 16.9367,Z 124,A 4.4664,B 24.9472,C -1.6783,E1 25.1581,E2 441.5903} C_DIS
LIN {X 118.4696,Y 19.8391,Z 124,A 5.8729,B 24.9469,C -1.6831,E1 25.1574,E2 440.1809} C_DIS
LIN {X 117.9471,Y 22.7405,Z 124,A 7.2568,B 24.9467,C -1.6864,E1 25.1567,E2 438.7972} C_DIS
LIN {X 117.3535,Y 25.6283,Z 124,A 8.6538,B 24.9465,C -1.6904,E1 25.1559,E2 437.3989} C_DIS
LIN {X 116.7035,Y 28.4417,Z 124,A 10.0478,B 24.9461,C -1.6956,E1 25.155,E2 436.0009} C_DIS
LIN {X 115.9546,Y 31.3556,Z 124,A 11.4475,B 24.946,C -1.6983,E1 25.154,E2 434.6028} C_DIS
LIN {X 115.1559,Y 34.1725,Z 124,A 12.8393,B 24.9457,C -1.7023,E1 25.1529,E2 433.2094} C_DIS
LIN {X 114.2764,Y 37.0075,Z 124,A 14.2547,B 24.9454,C -1.7066,E1 25.1517,E2 431.792} C_DIS
LIN {X 113.3337,Y 39.8008,Z 124,A 15.6518,B 24.9452,C -1.7104,E1 25.1505,E2 430.3937} C_DIS
LIN {X 112.3228,Y 42.5702,Z 124,A 17.0492,B 24.9449,C -1.7142,E1 25.1491,E2 428.9953} C_DIS
LIN {X 111.2443,Y 45.3139,Z 124,A 18.4466,B 24.9447,C -1.7179,E1 25.1476,E2 427.5968} C_DIS
LIN {X 110.0987,Y 48.0303,Z 124,A 19.8441,B 24.9445,C -1.7216,E1 25.1461,E2 426.1983} C_DIS
LIN {X 108.8868,Y 50.7178,Z 124,A 21.2416,B 24.9442,C -1.7252,E1 25.1445,E2 424.7998} C_DIS
LIN {X 107.6094,Y 53.3748,Z 124,A 22.6395,B 24.944,C -1.7288,E1 25.1428,E2 423.4009} C_DIS
LIN {X 106.2671,Y 55.9996,Z 124,A 24.0376,B 24.9438,C -1.7323,E1 25.141,E2 422.0019} C_DIS
LIN {X 104.8608,Y 58.5906,Z 124,A 25.4225,B 24.9436,C -1.7352,E1 25.1391,E2 420.6176} C_DIS
LIN {X 103.3928,Y 61.1439,Z 124,A 26.8198,B 24.9433,C -1.7386,E1 25.1371,E2 419.2192} C_DIS
LIN {X 101.8596,Y 63.6653,Z 124,A 28.2659,B 24.943,C -1.7443,E1 25.135,E2 417.7672} C_DIS
LIN {X 99.8774,Y 66.736,Z 124,A 29.9657,B 24.9428,C -1.7467,E1 25.1324,E2 416.0703} C_DIS
LIN {X 98.0222,Y 69.4296,Z 124,A 31.3792,B 24.943,C -1.7436,E1 25.1302,E2 414.671} C_DIS
Enddeposition()
END
